C01810=1159.074,186.001,-60.182,-178.162,7.026,148.772
C01811=1159.078,185.752,-60.160,-178.165,7.023,148.772
C01812=1159.083,185.503,-60.136,-178.168,7.021,148.772
C01813=1159.087,185.254,-60.113,-178.170,7.019,148.772
C01814=1159.092,185.005,-60.089,-178.174,7.017,148.773
C01815=1159.097,184.757,-60.067,-178.176,7.015,148.773
C01816=1159.101,184.508,-60.044,-178.178,7.013,148.773
C01817=1159.107,184.238,-60.019,-178.182,7.010,148.774
C01818=1159.112,183.969,-59.994,-178.185,7.008,148.774
C01819=1159.117,183.699,-59.969,-178.187,7.006,148.774
C01820=1159.121,183.429,-59.943,-178.190,7.003,148.774
C01821=1159.127,183.180,-59.921,-178.193,7.001,148.775
C01822=1159.131,182.932,-59.898,-178.196,6.999,148.775
C01823=1159.135,182.683,-59.875,-178.199,6.997,148.775
C01824=1159.140,182.433,-59.851,-178.201,6.995,148.776
C01825=1159.144,182.185,-59.829,-178.205,6.992,148.776
C01826=1159.149,181.936,-59.806,-178.207,6.991,148.776
C01827=1159.154,181.687,-59.783,-178.209,6.989,148.776
C01828=1159.158,181.438,-59.760,-178.212,6.987,148.777
C01829=1159.163,181.189,-59.737,-178.215,6.984,148.777
C01830=1159.168,180.940,-59.713,-178.218,6.982,148.777
C01831=1159.172,180.692,-59.691,-178.220,6.980,148.778
C01832=1159.177,180.442,-59.668,-178.224,6.978,148.778
C01833=1159.181,180.194,-59.646,-178.226,6.976,148.778
C01834=1159.186,179.945,-59.622,-178.229,6.974,148.778
C01835=1159.190,179.697,-59.600,-178.232,6.971,148.779
C01836=1159.195,179.447,-59.577,-178.234,6.970,148.779
C01837=1159.200,179.198,-59.554,-178.237,6.968,148.780
C01838=1159.204,178.949,-59.531,-178.240,6.965,148.780
C01839=1159.210,178.700,-59.509,-178.243,6.963,148.780
C01840=1159.214,178.451,-59.486,-178.245,6.961,148.780
C01841=1159.218,178.202,-59.463,-178.248,6.960,148.781
C01842=1159.223,177.953,-59.441,-178.251,6.957,148.781
C01843=1159.228,177.705,-59.418,-178.254,6.955,148.781
C01844=1159.232,177.455,-59.396,-178.256,6.953,148.782
C01845=1159.237,177.206,-59.372,-178.259,6.951,148.782
C01846=1159.241,176.958,-59.349,-178.262,6.949,148.782
C01847=1159.246,176.709,-59.327,-178.264,6.947,148.782
C01848=1159.250,176.460,-59.304,-178.268,6.944,148.783
C01849=1159.255,176.210,-59.282,-178.270,6.943,148.783
C01850=1159.260,175.962,-59.259,-178.273,6.940,148.783
C01851=1159.265,175.713,-59.237,-178.275,6.939,148.784
C01852=1159.269,175.464,-59.214,-178.278,6.936,148.784
C01853=1159.275,175.215,-59.192,-178.281,6.934,148.784
C01854=1159.278,174.966,-59.169,-178.284,6.933,148.785
C01855=1159.283,174.717,-59.147,-178.286,6.931,148.785
C01856=1159.288,174.469,-59.124,-178.289,6.928,148.785
C01857=1159.292,174.219,-59.102,-178.292,6.926,148.786
C01858=1159.297,173.970,-59.079,-178.295,6.924,148.786
C01859=1159.302,173.722,-59.057,-178.298,6.922,148.786
C01860=1159.306,173.472,-59.035,-178.300,6.920,148.786
C01861=1159.311,173.224,-59.012,-178.303,6.918,148.787
C01862=1159.316,172.975,-58.990,-178.306,6.916,148.787
C01863=1159.320,172.726,-58.966,-178.309,6.914,148.788
C01864=1159.325,172.477,-58.945,-178.311,6.912,148.788
C01865=1159.330,172.228,-58.923,-178.314,6.910,148.788
C01866=1159.334,171.979,-58.899,-178.316,6.908,148.788
C01867=1159.339,171.730,-58.878,-178.320,6.906,148.789
C01868=1159.343,171.481,-58.856,-178.322,6.904,148.789
C01869=1159.349,171.232,-58.833,-178.325,6.902,148.789
C01870=1159.353,170.983,-58.811,-178.327,6.900,148.790
C01871=1159.358,170.734,-58.789,-178.331,6.897,148.790
C01872=1159.363,170.485,-58.766,-178.333,6.896,148.790
C01873=1159.367,170.236,-58.743,-178.336,6.894,148.791
C01874=1159.372,169.987,-58.722,-178.338,6.892,148.791
C01875=1159.376,169.738,-58.700,-178.341,6.890,148.791
C01876=1159.382,169.489,-58.677,-178.344,6.888,148.792
C01877=1159.386,169.240,-58.655,-178.347,6.886,148.792
C01878=1159.390,168.992,-58.633,-178.350,6.884,148.792
C01879=1159.395,168.742,-58.611,-178.352,6.882,148.793
C01880=1159.400,168.493,-58.589,-178.355,6.879,148.793
C01881=1159.405,168.244,-58.567,-178.358,6.878,148.793
C01882=1159.409,167.996,-58.544,-178.360,6.876,148.794
C01883=1159.413,167.747,-58.522,-178.363,6.874,148.794
C01884=1159.419,167.498,-58.500,-178.366,6.872,148.794
C01885=1159.423,167.248,-58.478,-178.369,6.870,148.795
C01886=1159.428,167.000,-58.456,-178.371,6.868,148.795
C01887=1159.432,166.750,-58.434,-178.374,6.866,148.795
C01888=1159.437,166.502,-58.412,-178.377,6.864,148.796
C01889=1159.442,166.252,-58.390,-178.380,6.862,148.796
C01890=1159.447,166.003,-58.368,-178.383,6.860,148.796
C01891=1159.451,165.754,-58.346,-178.385,6.858,148.797
C01892=1159.456,165.505,-58.324,-178.388,6.856,148.797
C01893=1159.461,165.256,-58.302,-178.390,6.854,148.797
C01894=1159.465,165.007,-58.281,-178.394,6.852,148.798
C01895=1159.470,164.758,-58.259,-178.396,6.850,148.798
C01896=1159.475,164.509,-58.237,-178.399,6.848,148.798
C01897=1159.479,164.260,-58.215,-178.402,6.847,148.799
C01898=1159.484,164.011,-58.193,-178.404,6.845,148.799
C01899=1159.489,163.762,-58.171,-178.407,6.842,148.799
C01900=1159.494,163.513,-58.149,-178.410,6.840,148.800
C01901=1159.498,163.264,-58.127,-178.413,6.838,148.800
C01902=1159.503,163.015,-58.105,-178.415,6.837,148.800
C01903=1159.508,162.767,-58.083,-178.418,6.835,148.801
C01904=1159.512,162.517,-58.061,-178.421,6.833,148.801
C01905=1159.517,162.269,-58.040,-178.424,6.831,148.801
C01906=1159.521,162.019,-58.018,-178.427,6.829,148.802
C01907=1159.526,161.771,-57.996,-178.429,6.827,148.802
C01908=1159.531,161.522,-57.974,-178.432,6.825,148.802
C01909=1159.535,161.272,-57.953,-178.434,6.823,148.803
C01910=1159.540,161.023,-57.931,-178.437,6.821,148.803
C01911=1159.544,160.774,-57.909,-178.440,6.819,148.803
C01912=1159.549,160.525,-57.888,-178.443,6.817,148.804
C01913=1159.554,160.277,-57.866,-178.446,6.816,148.804
C01914=1159.559,160.027,-57.845,-178.448,6.814,148.805
C01915=1159.564,159.778,-57.823,-178.451,6.812,148.805
C01916=1159.568,159.529,-57.801,-178.453,6.810,148.805
C01917=1159.573,159.280,-57.779,-178.456,6.807,148.805
C01918=1159.578,159.031,-57.758,-178.459,6.806,148.806
C01919=1159.582,158.783,-57.737,-178.462,6.804,148.806
C01920=1159.586,158.533,-57.715,-178.465,6.802,148.807
C01921=1159.592,158.264,-57.692,-178.467,6.800,148.807
C01922=1159.596,157.995,-57.668,-178.471,6.798,148.807
C01923=1159.602,157.726,-57.645,-178.473,6.796,148.808
C01924=1159.607,157.458,-57.622,-178.477,6.794,148.808
C01925=1159.611,157.208,-57.600,-178.479,6.792,148.808
C01926=1159.616,156.959,-57.579,-178.482,6.790,148.809
C01927=1159.621,156.710,-57.558,-178.485,6.788,148.809
C01928=1159.626,156.461,-57.536,-178.487,6.787,148.809
C01929=1159.631,156.212,-57.515,-178.490,6.785,148.810
C01930=1159.636,155.963,-57.493,-178.493,6.782,148.810
C01931=1159.640,155.714,-57.472,-178.496,6.781,148.811
C01932=1159.644,155.465,-57.451,-178.499,6.779,148.811
C01933=1159.649,155.216,-57.429,-178.501,6.777,148.811
C01934=1159.654,154.967,-57.408,-178.504,6.775,148.812
C01935=1159.659,154.718,-57.386,-178.506,6.773,148.812
C01936=1159.663,154.469,-57.366,-178.509,6.772,148.812
C01937=1159.668,154.220,-57.344,-178.512,6.770,148.813
C01938=1159.673,153.971,-57.323,-178.514,6.768,148.813
C01939=1159.677,153.722,-57.301,-178.518,6.766,148.813
C01940=1159.683,153.472,-57.280,-178.520,6.764,148.814
C01941=1159.687,153.224,-57.259,-178.523,6.762,148.814
C01942=1159.692,152.975,-57.238,-178.526,6.760,148.815
C01943=1159.697,152.726,-57.216,-178.528,6.759,148.815
C01944=1159.701,152.476,-57.195,-178.531,6.757,148.815
C01945=1159.706,152.227,-57.174,-178.534,6.755,148.816
C01946=1159.711,151.978,-57.153,-178.537,6.753,148.816
C01947=1159.716,151.729,-57.132,-178.539,6.752,148.816
C01948=1159.720,151.481,-57.111,-178.543,6.749,148.817
C01949=1159.725,151.231,-57.089,-178.545,6.747,148.817
C01950=1159.730,150.982,-57.068,-178.548,6.746,148.818
C01951=1159.735,150.733,-57.047,-178.551,6.744,148.818
C01952=1159.739,150.484,-57.026,-178.553,6.742,148.818
C01953=1159.744,150.235,-57.005,-178.556,6.740,148.819
C01954=1159.748,149.985,-56.983,-178.559,6.739,148.819
C01955=1159.753,149.737,-56.963,-178.561,6.737,148.819
C01956=1159.758,149.487,-56.942,-178.564,6.735,148.820
C01957=1159.762,149.239,-56.921,-178.566,6.733,148.820
C01958=1159.767,148.990,-56.900,-178.569,6.731,148.820
C01959=1159.773,148.740,-56.879,-178.572,6.729,148.821
C01960=1159.777,148.492,-56.858,-178.575,6.727,148.821
C01961=1159.781,148.242,-56.837,-178.578,6.725,148.822
C01962=1159.786,147.993,-56.816,-178.581,6.724,148.822
C01963=1159.791,147.744,-56.795,-178.583,6.722,148.822
C01964=1159.796,147.495,-56.774,-178.586,6.720,148.823
C01965=1159.800,147.246,-56.753,-178.589,6.719,148.823
C01966=1159.805,146.997,-56.732,-178.591,6.717,148.823
C01967=1159.810,146.748,-56.712,-178.594,6.715,148.824
C01968=1159.815,146.499,-56.691,-178.597,6.713,148.824
C01969=1159.819,146.250,-56.670,-178.599,6.712,148.825
C01970=1159.824,146.001,-56.648,-178.602,6.710,148.825
C01971=1159.829,145.751,-56.627,-178.605,6.708,148.825
C01972=1159.833,145.502,-56.607,-178.608,6.706,148.826
C01973=1159.838,145.253,-56.586,-178.610,6.705,148.826
C01974=1159.843,145.004,-56.566,-178.613,6.703,148.827
C01975=1159.848,144.755,-56.545,-178.616,6.700,148.827
C01976=1159.853,144.506,-56.524,-178.619,6.699,148.827
C01977=1159.858,144.257,-56.503,-178.622,6.697,148.828
C01978=1159.862,144.008,-56.483,-178.624,6.695,148.828
C01979=1159.867,143.759,-56.463,-178.627,6.693,148.828
C01980=1159.872,143.510,-56.442,-178.630,6.692,148.829
C01981=1159.876,143.261,-56.421,-178.632,6.690,148.829
C01982=1159.881,143.011,-56.400,-178.635,6.688,148.830
C01983=1159.886,142.762,-56.380,-178.638,6.687,148.830
C01984=1159.891,142.513,-56.359,-178.641,6.685,148.830
C01985=1159.895,142.264,-56.339,-178.643,6.683,148.831
C01986=1159.900,142.015,-56.318,-178.646,6.681,148.831
C01987=1159.905,141.766,-56.297,-178.649,6.680,148.832
C01988=1159.909,141.517,-56.277,-178.651,6.678,148.832
C01989=1159.915,141.268,-56.256,-178.654,6.676,148.832
C01990=1159.919,141.019,-56.236,-178.657,6.674,148.833
C01991=1159.923,140.770,-56.215,-178.660,6.673,148.833
C01992=1159.929,140.521,-56.194,-178.662,6.671,148.833
C01993=1159.933,140.272,-56.174,-178.665,6.670,148.834
C01994=1159.938,140.023,-56.154,-178.668,6.668,148.834
C01995=1159.943,139.773,-56.133,-178.671,6.666,148.835
C01996=1159.947,139.524,-56.113,-178.674,6.664,148.835
C01997=1159.952,139.275,-56.093,-178.676,6.663,148.836
C01998=1159.957,139.026,-56.072,-178.679,6.661,148.836
C01999=1159.962,138.777,-56.051,-178.682,6.659,148.836
C02000=1159.966,138.528,-56.031,-178.684,6.658,148.837
C02001=1159.971,138.278,-56.010,-178.687,6.656,148.837
C02002=1159.976,138.029,-55.990,-178.690,6.654,148.838
C02003=1159.980,137.780,-55.970,-178.692,6.652,148.838
C02004=1159.985,137.531,-55.949,-178.695,6.651,148.838
C02005=1159.990,137.282,-55.928,-178.698,6.649,148.839
C02006=1159.995,137.032,-55.909,-178.701,6.647,148.839
C02007=1159.999,136.783,-55.888,-178.703,6.645,148.840
C02008=1160.004,136.534,-55.868,-178.706,6.644,148.840
C02009=1160.009,136.286,-55.847,-178.709,6.642,148.840
C02010=1160.014,136.036,-55.828,-178.711,6.640,148.841
C02011=1160.018,135.787,-55.807,-178.714,6.639,148.841
C02012=1160.023,135.538,-55.787,-178.717,6.637,148.841
C02013=1160.028,135.288,-55.767,-178.720,6.635,148.842
C02014=1160.033,135.039,-55.746,-178.723,6.634,148.842
C02015=1160.037,134.791,-55.726,-178.725,6.632,148.843
C02016=1160.042,134.541,-55.706,-178.728,6.630,148.843
C02017=1160.047,134.293,-55.686,-178.731,6.629,148.844
C02018=1160.052,134.043,-55.665,-178.734,6.627,148.844
C02019=1160.057,133.794,-55.646,-178.736,6.625,148.844
C02020=1160.061,133.545,-55.625,-178.739,6.623,148.845
C02021=1160.066,133.295,-55.606,-178.742,6.622,148.845
C02022=1160.071,133.046,-55.585,-178.744,6.620,148.846
C02023=1160.075,132.797,-55.566,-178.747,6.618,148.846
C02024=1160.081,132.548,-55.545,-178.750,6.616,148.846
C02025=1160.086,132.280,-55.524,-178.753,6.615,148.847
C02026=1160.091,132.012,-55.502,-178.756,6.613,148.847
C02027=1160.096,131.743,-55.481,-178.758,6.612,148.848
C02028=1160.101,131.474,-55.460,-178.761,6.610,148.848
C02029=1160.106,131.225,-55.439,-178.764,6.608,148.849
C02030=1160.110,130.975,-55.419,-178.767,6.607,148.849
C02031=1160.116,130.726,-55.399,-178.770,6.605,148.850
C02032=1160.121,130.477,-55.379,-178.772,6.603,148.850
C02033=1160.125,130.228,-55.359,-178.775,6.602,148.850
C02034=1160.130,129.979,-55.339,-178.778,6.600,148.851
C02035=1160.135,129.730,-55.319,-178.781,6.598,148.851
C02036=1160.139,129.480,-55.299,-178.783,6.597,148.852
C02037=1160.145,129.231,-55.280,-178.786,6.595,148.852
C02038=1160.149,128.982,-55.259,-178.789,6.593,148.852
C02039=1160.154,128.733,-55.240,-178.791,6.591,148.853
C02040=1160.159,128.483,-55.220,-178.795,6.590,148.853
C02041=1160.164,128.235,-55.200,-178.797,6.588,148.854
C02042=1160.168,127.986,-55.181,-178.800,6.587,148.854
C02043=1160.173,127.737,-55.160,-178.803,6.585,148.855
C02044=1160.177,127.487,-55.140,-178.805,6.584,148.855
C02045=1160.183,127.238,-55.121,-178.808,6.582,148.855
C02046=1160.188,126.989,-55.102,-178.810,6.581,148.856
C02047=1160.192,126.740,-55.081,-178.813,6.579,148.856
C02048=1160.197,126.491,-55.062,-178.816,6.577,148.857
C02049=1160.202,126.241,-55.042,-178.819,6.576,148.857
C02050=1160.207,125.992,-55.022,-178.822,6.574,148.858
C02051=1160.211,125.743,-55.003,-178.824,6.572,148.858
C02052=1160.216,125.494,-54.984,-178.827,6.571,148.858
C02053=1160.221,125.245,-54.964,-178.830,6.569,148.859
C02054=1160.225,124.996,-54.943,-178.832,6.567,148.859
C02055=1160.230,124.747,-54.924,-178.835,6.566,148.860
C02056=1160.235,124.497,-54.905,-178.838,6.565,148.860
C02057=1160.240,124.248,-54.885,-178.840,6.563,148.861
C02058=1160.245,123.999,-54.866,-178.843,6.561,148.861
C02059=1160.250,123.749,-54.846,-178.846,6.560,148.861
C02060=1160.254,123.501,-54.826,-178.849,6.558,148.862
C02061=1160.259,123.252,-54.807,-178.851,6.556,148.862
C02062=1160.264,123.002,-54.787,-178.854,6.555,148.863
C02063=1160.269,122.753,-54.768,-178.857,6.553,148.863
C02064=1160.274,122.504,-54.748,-178.860,6.551,148.864
C02065=1160.279,122.254,-54.729,-178.862,6.551,148.864
C02066=1160.283,122.005,-54.710,-178.865,6.549,148.864
C02067=1160.288,121.756,-54.690,-178.868,6.547,148.865
C02068=1160.293,121.506,-54.671,-178.870,6.545,148.865
C02069=1160.298,121.258,-54.651,-178.873,6.544,148.866
C02070=1160.302,121.009,-54.631,-178.876,6.542,148.866
C02071=1160.306,120.759,-54.612,-178.879,6.541,148.867
C02072=1160.312,120.510,-54.593,-178.882,6.539,148.867
C02073=1160.317,120.261,-54.573,-178.884,6.538,148.867
C02074=1160.322,120.012,-54.554,-178.886,6.536,148.868
C02075=1160.326,119.763,-54.535,-178.889,6.535,148.868
C02076=1160.331,119.513,-54.515,-178.892,6.533,148.869
C02077=1160.336,119.264,-54.496,-178.895,6.532,148.869
C02078=1160.341,119.015,-54.476,-178.898,6.530,148.870
C02079=1160.345,118.766,-54.457,-178.900,6.528,148.870
C02080=1160.350,118.516,-54.438,-178.903,6.527,148.870
C02081=1160.356,118.267,-54.419,-178.905,6.525,148.871
C02082=1160.360,118.018,-54.400,-178.909,6.524,148.871
C02083=1160.365,117.769,-54.381,-178.911,6.522,148.872
C02084=1160.370,117.519,-54.361,-178.914,6.521,148.872
C02085=1160.374,117.270,-54.342,-178.917,6.519,148.873
C02086=1160.379,117.021,-54.323,-178.919,6.517,148.873
C02087=1160.384,116.772,-54.303,-178.922,6.516,148.874
C02088=1160.389,116.523,-54.284,-178.925,6.515,148.874
C02089=1160.394,116.273,-54.265,-178.927,6.513,148.875
C02090=1160.399,116.024,-54.246,-178.930,6.512,148.875
C02091=1160.403,115.775,-54.227,-178.933,6.510,148.875
C02092=1160.408,115.526,-54.208,-178.936,6.508,148.876
C02093=1160.413,115.276,-54.188,-178.938,6.508,148.876
C02094=1160.418,115.028,-54.169,-178.941,6.506,148.877
C02095=1160.423,114.778,-54.150,-178.944,6.504,148.877
C02096=1160.427,114.529,-54.132,-178.946,6.502,148.878
C02097=1160.432,114.280,-54.112,-178.949,6.501,148.878
C02098=1160.437,114.031,-54.093,-178.952,6.499,148.879
C02099=1160.442,113.781,-54.074,-178.954,6.499,148.879
C02100=1160.447,113.532,-54.055,-178.957,6.497,148.879
C02101=1160.452,113.283,-54.036,-178.960,6.495,148.880
C02102=1160.457,113.033,-54.018,-178.963,6.493,148.880
C02103=1160.461,112.785,-53.999,-178.966,6.492,148.881
C02104=1160.466,112.535,-53.979,-178.968,6.490,148.881
C02105=1160.472,112.286,-53.961,-178.971,6.489,148.882
C02106=1160.476,112.036,-53.942,-178.973,6.488,148.882
C02107=1160.481,111.787,-53.922,-178.976,6.486,148.883
C02108=1160.485,111.538,-53.904,-178.979,6.485,148.883
C02109=1160.491,111.289,-53.885,-178.982,6.483,148.884
C02110=1160.495,111.040,-53.866,-178.984,6.482,148.884
C02111=1160.500,110.790,-53.847,-178.987,6.480,148.884
C02112=1160.505,110.541,-53.828,-178.990,6.479,148.885
C02113=1160.510,110.291,-53.809,-178.993,6.477,148.885
C02114=1160.515,110.043,-53.791,-178.995,6.476,148.886
C02115=1160.519,109.794,-53.772,-178.998,6.475,148.886
C02116=1160.524,109.544,-53.753,-179.000,6.473,148.887
C02117=1160.529,109.295,-53.734,-179.004,6.472,148.887
C02118=1160.534,109.045,-53.715,-179.006,6.470,148.888
C02119=1160.539,108.797,-53.697,-179.009,6.468,148.888
C02120=1160.544,108.547,-53.678,-179.011,6.467,148.888
C02121=1160.548,108.298,-53.659,-179.014,6.466,148.889
C02122=1160.553,108.049,-53.641,-179.017,6.464,148.890
C02123=1160.558,107.800,-53.622,-179.020,6.463,148.890
C02124=1160.563,107.550,-53.603,-179.022,6.462,148.890
C02125=1160.568,107.301,-53.584,-179.025,6.460,148.891
C02126=1160.572,107.051,-53.566,-179.028,6.459,148.891
C02127=1160.577,106.803,-53.547,-179.031,6.457,148.892
C02128=1160.583,106.553,-53.529,-179.033,6.455,148.892
C02129=1160.588,106.285,-53.509,-179.036,6.454,148.893
C02130=1160.593,106.016,-53.488,-179.039,6.452,148.893
C02131=1160.598,105.748,-53.469,-179.042,6.450,148.894
C02132=1160.604,105.479,-53.449,-179.045,6.449,148.894
C02133=1160.608,105.230,-53.430,-179.047,6.448,148.895
C02134=1160.612,104.981,-53.412,-179.050,6.447,148.895
C02135=1160.618,104.732,-53.393,-179.053,6.445,148.896
C02136=1160.623,104.483,-53.374,-179.056,6.443,148.896
C02137=1160.627,104.233,-53.356,-179.058,6.443,148.897
C02138=1160.633,103.984,-53.337,-179.061,6.441,148.897
C02139=1160.637,103.735,-53.319,-179.063,6.439,148.897
C02140=1160.642,103.485,-53.300,-179.067,6.438,148.898
C02141=1160.647,103.236,-53.282,-179.069,6.437,148.898
C02142=1160.652,102.987,-53.263,-179.071,6.435,148.899
C02143=1160.657,102.738,-53.245,-179.075,6.434,148.900
C02144=1160.661,102.488,-53.227,-179.077,6.432,148.900
C02145=1160.667,102.239,-53.208,-179.080,6.431,148.900
C02146=1160.671,101.990,-53.189,-179.082,6.430,148.901
C02147=1160.676,101.741,-53.172,-179.085,6.428,148.901
C02148=1160.681,101.491,-53.153,-179.088,6.427,148.902
C02149=1160.685,101.242,-53.135,-179.090,6.426,148.902
C02150=1160.691,100.993,-53.116,-179.093,6.424,148.903
C02151=1160.696,100.744,-53.098,-179.096,6.423,148.903
C02152=1160.700,100.494,-53.080,-179.098,6.422,148.904
C02153=1160.705,100.245,-53.062,-179.101,6.420,148.904
C02154=1160.710,99.996,-53.044,-179.104,6.418,148.905
C02155=1160.716,99.746,-53.025,-179.107,6.417,148.905
C02156=1160.720,99.498,-53.006,-179.109,6.416,148.906
C02157=1160.724,99.248,-52.988,-179.112,6.414,148.906
C02158=1160.729,98.998,-52.970,-179.115,6.413,148.907
C02159=1160.734,98.749,-52.952,-179.118,6.411,148.907
C02160=1160.739,98.500,-52.934,-179.120,6.410,148.907
C02161=1160.744,98.251,-52.916,-179.123,6.409,148.908
C02162=1160.749,98.001,-52.897,-179.126,6.407,148.909
C02163=1160.754,97.752,-52.879,-179.128,6.407,148.909
C02164=1160.759,97.502,-52.861,-179.131,6.405,148.909
C02165=1160.764,97.253,-52.843,-179.134,6.404,148.910
C02166=1160.769,97.004,-52.825,-179.136,6.403,148.910
C02167=1160.774,96.755,-52.807,-179.139,6.401,148.911
C02168=1160.778,96.505,-52.789,-179.142,6.399,148.911
C02169=1160.783,96.256,-52.771,-179.145,6.398,148.912
C02170=1160.788,96.007,-52.753,-179.147,6.397,148.912
C02171=1160.793,95.757,-52.735,-179.150,6.395,148.913
C02172=1160.798,95.508,-52.717,-179.153,6.394,148.913
C02173=1160.803,95.259,-52.699,-179.155,6.393,148.914
C02174=1160.807,95.010,-52.681,-179.158,6.391,148.914
C02175=1160.812,94.761,-52.663,-179.160,6.390,148.915
C02176=1160.817,94.511,-52.645,-179.163,6.389,148.915
C02177=1160.822,94.261,-52.626,-179.166,6.387,148.916
C02178=1160.827,94.012,-52.608,-179.169,6.386,148.916
C02179=1160.832,93.763,-52.590,-179.172,6.384,148.917
C02180=1160.837,93.514,-52.572,-179.174,6.384,148.917
C02181=1160.842,93.265,-52.554,-179.177,6.382,148.918
C02182=1160.846,93.016,-52.537,-179.180,6.381,148.918
C02183=1160.851,92.766,-52.520,-179.182,6.380,148.919
C02184=1160.856,92.517,-52.502,-179.185,6.378,148.919
C02185=1160.861,92.268,-52.484,-179.187,6.376,148.919
C02186=1160.866,92.019,-52.466,-179.190,6.376,148.920
C02187=1160.870,91.769,-52.447,-179.193,6.374,148.921
C02188=1160.875,91.519,-52.429,-179.195,6.372,148.921
C02189=1160.881,91.270,-52.412,-179.198,6.372,148.922
C02190=1160.885,91.021,-52.394,-179.201,6.370,148.922
C02191=1160.890,90.771,-52.376,-179.204,6.368,148.922
C02192=1160.895,90.522,-52.358,-179.206,6.368,148.923
C02193=1160.901,90.272,-52.341,-179.209,6.366,148.924
C02194=1160.905,90.023,-52.323,-179.212,6.364,148.924
C02195=1160.910,89.774,-52.305,-179.214,6.364,148.925
C02196=1160.915,89.525,-52.287,-179.217,6.362,148.925
C02197=1160.920,89.275,-52.270,-179.220,6.361,148.925
C02198=1160.925,89.026,-52.252,-179.222,6.360,148.926
C02199=1160.930,88.777,-52.234,-179.225,6.358,148.926
C02200=1160.935,88.527,-52.217,-179.227,6.357,148.927
C02201=1160.940,88.278,-52.199,-179.230,6.356,148.928
C02202=1160.945,88.029,-52.181,-179.233,6.354,148.928
C02203=1160.949,87.779,-52.164,-179.235,6.354,148.928
C02204=1160.954,87.530,-52.146,-179.239,6.352,148.929
C02205=1160.959,87.281,-52.128,-179.241,6.351,148.929
C02206=1160.964,87.031,-52.111,-179.243,6.350,148.930
C02207=1160.969,86.782,-52.093,-179.247,6.348,148.931
C02208=1160.973,86.533,-52.076,-179.249,6.347,148.931
C02209=1160.978,86.283,-52.058,-179.251,6.346,148.931
C02210=1160.983,86.034,-52.041,-179.255,6.344,148.932
C02211=1160.989,85.784,-52.023,-179.257,6.344,148.932
C02212=1160.993,85.535,-52.005,-179.260,6.342,148.933
C02213=1160.998,85.286,-51.988,-179.263,6.341,148.934
C02214=1161.003,85.037,-51.971,-179.265,6.340,148.934
C02215=1161.008,84.787,-51.953,-179.268,6.338,148.934
C02216=1161.014,84.538,-51.936,-179.271,6.337,148.935
C02217=1161.018,84.289,-51.918,-179.273,6.336,148.935
C02218=1161.023,84.040,-51.901,-179.276,6.334,148.936
C02219=1161.028,83.790,-51.883,-179.278,6.334,148.937
C02220=1161.033,83.541,-51.866,-179.281,6.332,148.937
C02221=1161.037,83.292,-51.848,-179.284,6.330,148.937
C02222=1161.042,83.042,-51.831,-179.286,6.330,148.938
C02223=1161.047,82.793,-51.813,-179.289,6.328,148.938
C02224=1161.052,82.543,-51.797,-179.292,6.327,148.939
C02225=1161.057,82.294,-51.779,-179.295,6.326,148.940
C02226=1161.062,82.044,-51.761,-179.297,6.324,148.940
C02227=1161.067,81.796,-51.745,-179.300,6.324,148.941
C02228=1161.072,81.546,-51.727,-179.303,6.322,148.941
C02229=1161.077,81.297,-51.710,-179.305,6.321,148.941
C02230=1161.081,81.048,-51.692,-179.308,6.320,148.942
C02231=1161.087,80.798,-51.675,-179.311,6.318,148.943
C02232=1161.092,80.548,-51.658,-179.313,6.317,148.943
C02233=1161.097,80.280,-51.640,-179.316,6.316,148.944
C02234=1161.102,80.012,-51.621,-179.319,6.314,148.944
C02235=1161.108,79.743,-51.602,-179.322,6.313,148.945
C02236=1161.113,79.475,-51.584,-179.325,6.312,148.945
C02237=1161.118,79.226,-51.567,-179.327,6.311,148.946
C02238=1161.123,78.976,-51.549,-179.330,6.309,148.946
C02239=1161.127,78.727,-51.532,-179.333,6.308,148.947
C02240=1161.133,78.477,-51.515,-179.335,6.307,148.947
C02241=1161.137,78.228,-51.498,-179.338,6.306,148.948
C02242=1161.143,77.979,-51.481,-179.341,6.305,148.948
C02243=1161.147,77.730,-51.464,-179.343,6.304,148.949
C02244=1161.152,77.480,-51.447,-179.346,6.302,148.949
C02245=1161.157,77.231,-51.429,-179.349,6.301,148.950
C02246=1161.162,76.981,-51.412,-179.351,6.300,148.950
C02247=1161.168,76.732,-51.395,-179.354,6.298,148.951
C02248=1161.172,76.483,-51.379,-179.356,6.298,148.951
C02249=1161.177,76.233,-51.361,-179.359,6.296,148.952
C02250=1161.181,75.984,-51.344,-179.362,6.295,148.952
C02251=1161.187,75.734,-51.327,-179.365,6.294,148.953
C02252=1161.192,75.485,-51.310,-179.367,6.293,148.954
C02253=1161.197,75.236,-51.293,-179.370,6.291,148.954
C02254=1161.201,74.986,-51.277,-179.373,6.290,148.954
C02255=1161.206,74.737,-51.260,-179.375,6.289,148.955
C02256=1161.211,74.488,-51.242,-179.378,6.288,148.955
C02257=1161.216,74.239,-51.226,-179.381,6.287,148.956
C02258=1161.221,73.989,-51.208,-179.383,6.285,148.957
C02259=1161.226,73.739,-51.192,-179.386,6.285,148.957
C02260=1161.231,73.490,-51.175,-179.389,6.283,148.958
C02261=1161.236,73.241,-51.158,-179.391,6.282,148.958
C02262=1161.241,72.991,-51.141,-179.394,6.281,148.959
C02263=1161.246,72.742,-51.124,-179.397,6.279,148.959
C02264=1161.251,72.493,-51.108,-179.399,6.278,148.960
C02265=1161.256,72.243,-51.091,-179.402,6.277,148.960
C02266=1161.260,71.993,-51.074,-179.404,6.276,148.961
C02267=1161.266,71.744,-51.057,-179.408,6.275,148.961
C02268=1161.271,71.495,-51.040,-179.410,6.274,148.962
C02269=1161.275,71.245,-51.024,-179.412,6.272,148.962
C02270=1161.281,70.996,-51.007,-179.415,6.272,148.963
C02271=1161.285,70.747,-50.990,-179.418,6.270,148.963
C02272=1161.290,70.497,-50.973,-179.420,6.270,148.964
C02273=1161.296,70.248,-50.957,-179.423,6.268,148.964
C02274=1161.300,69.999,-50.940,-179.425,6.267,148.965
C02275=1161.305,69.749,-50.923,-179.429,6.266,148.965
C02276=1161.311,69.500,-50.906,-179.431,6.265,148.966
C02277=1161.315,69.251,-50.890,-179.434,6.264,148.967
C02278=1161.320,69.001,-50.872,-179.436,6.263,148.967
C02279=1161.325,68.752,-50.856,-179.439,6.261,148.967
C02280=1161.330,68.503,-50.839,-179.441,6.261,148.968
C02281=1161.334,68.253,-50.823,-179.444,6.259,148.969
C02282=1161.340,68.004,-50.806,-179.447,6.258,148.969
C02283=1161.345,67.754,-50.790,-179.450,6.257,148.970
C02284=1161.349,67.504,-50.773,-179.452,6.256,148.970
C02285=1161.355,67.255,-50.756,-179.455,6.255,148.971
C02286=1161.360,67.006,-50.740,-179.457,6.254,148.971
C02287=1161.364,66.756,-50.723,-179.460,6.252,148.972
C02288=1161.369,66.508,-50.707,-179.462,6.252,148.972
C02289=1161.374,66.258,-50.691,-179.466,6.250,148.973
C02290=1161.380,66.008,-50.674,-179.468,6.249,148.973
C02291=1161.384,65.759,-50.657,-179.471,6.248,148.974
C02292=1161.389,65.509,-50.640,-179.473,6.247,148.974
C02293=1161.394,65.261,-50.624,-179.476,6.246,148.975
C02294=1161.399,65.010,-50.608,-179.479,6.245,148.976
C02295=1161.404,64.761,-50.591,-179.481,6.243,148.976
C02296=1161.409,64.512,-50.575,-179.484,6.243,148.977
C02297=1161.414,64.263,-50.559,-179.487,6.241,148.977
C02298=1161.419,64.013,-50.542,-179.489,6.240,148.977
C02299=1161.424,63.763,-50.525,-179.492,6.239,148.978
C02300=1161.429,63.515,-50.509,-179.494,6.238,148.979
C02301=1161.434,63.264,-50.493,-179.497,6.237,148.979
C02302=1161.439,63.016,-50.477,-179.500,6.236,148.980
C02303=1161.443,62.766,-50.460,-179.503,6.235,148.980
C02304=1161.449,62.517,-50.444,-179.505,6.234,148.981
C02305=1161.453,62.267,-50.428,-179.508,6.232,148.981
C02306=1161.459,62.018,-50.411,-179.510,6.232,148.982
C02307=1161.464,61.768,-50.395,-179.513,6.230,148.982
C02308=1161.469,61.519,-50.378,-179.516,6.229,148.983
C02309=1161.473,61.270,-50.362,-179.518,6.229,148.983
C02310=1161.478,61.020,-50.346,-179.521,6.227,148.984
C02311=1161.483,60.771,-50.330,-179.523,6.226,148.985
C02312=1161.488,60.521,-50.314,-179.526,6.225,148.985
C02313=1161.493,60.272,-50.297,-179.529,6.224,148.986
C02314=1161.498,60.022,-50.281,-179.531,6.223,148.986
C02315=1161.503,59.773,-50.265,-179.534,6.222,148.987
C02316=1161.508,59.524,-50.248,-179.537,6.220,148.987
C02317=1161.514,59.274,-50.232,-179.539,6.220,148.988
C02318=1161.519,59.025,-50.216,-179.542,6.218,148.988
C02319=1161.524,58.775,-50.200,-179.545,6.218,148.989
C02320=1161.529,58.526,-50.184,-179.547,6.217,148.989
C02321=1161.533,58.276,-50.168,-179.550,6.215,148.990
C02322=1161.538,58.027,-50.151,-179.552,6.215,148.990
C02323=1161.543,57.777,-50.135,-179.555,6.213,148.991
C02324=1161.548,57.529,-50.119,-179.558,6.213,148.992
C02325=1161.553,57.278,-50.103,-179.560,6.211,148.992
C02326=1161.558,57.030,-50.087,-179.563,6.210,148.993
C02327=1161.563,56.780,-50.071,-179.565,6.209,148.993
C02328=1161.568,56.530,-50.055,-179.568,6.208,148.994
C02329=1161.573,56.281,-50.039,-179.571,6.207,148.994
C02330=1161.578,56.031,-50.023,-179.574,6.206,148.995
C02331=1161.583,55.782,-50.007,-179.576,6.205,148.995
C02332=1161.588,55.532,-49.991,-179.579,6.203,148.996
C02333=1161.594,55.283,-49.975,-179.581,6.203,148.996
C02334=1161.598,55.033,-49.959,-179.583,6.202,148.997
C02335=1161.603,54.784,-49.943,-179.587,6.201,148.998
C02336=1161.608,54.536,-49.927,-179.589,6.200,148.998
C02337=1161.613,54.266,-49.910,-179.592,6.199,148.999
C02338=1161.618,53.998,-49.893,-179.595,6.197,148.999
C02339=1161.624,53.729,-49.876,-179.597,6.196,149.000
C02340=1161.629,53.461,-49.859,-179.601,6.195,149.000
C02341=1161.634,53.211,-49.843,-179.603,6.194,149.001
C02342=1161.640,52.961,-49.827,-179.606,6.193,149.001
C02343=1161.645,52.713,-49.811,-179.608,6.192,149.002
C02344=1161.649,52.463,-49.795,-179.611,6.192,149.003
C02345=1161.655,52.213,-49.779,-179.614,6.190,149.003
C02346=1161.660,51.964,-49.763,-179.616,6.190,149.004
C02347=1161.665,51.714,-49.747,-179.619,6.188,149.004
C02348=1161.669,51.465,-49.732,-179.622,6.187,149.005
C02349=1161.675,51.216,-49.717,-179.624,6.187,149.005
C02350=1161.679,50.966,-49.701,-179.627,6.185,149.006
C02351=1161.685,50.717,-49.684,-179.629,6.184,149.006
C02352=1161.690,50.467,-49.669,-179.632,6.183,149.007
C02353=1161.694,50.218,-49.653,-179.635,6.182,149.007
C02354=1161.699,49.968,-49.638,-179.637,6.181,149.008
C02355=1161.705,49.719,-49.622,-179.640,6.180,149.009
C02356=1161.709,49.469,-49.606,-179.642,6.179,149.009
C02357=1161.715,49.220,-49.590,-179.645,6.179,149.010
C02358=1161.719,48.971,-49.575,-179.648,6.177,149.010
C02359=1161.724,48.721,-49.559,-179.650,6.177,149.011
C02360=1161.729,48.471,-49.543,-179.653,6.175,149.011
C02361=1161.735,48.222,-49.528,-179.656,6.174,149.012
C02362=1161.740,47.972,-49.512,-179.658,6.174,149.012
C02363=1161.744,47.723,-49.496,-179.661,6.172,149.013
C02364=1161.749,47.474,-49.481,-179.663,6.171,149.013
C02365=1161.755,47.225,-49.465,-179.666,6.171,149.014
C02366=1161.759,46.975,-49.450,-179.668,6.169,149.015
C02367=1161.764,46.725,-49.434,-179.671,6.169,149.015
C02368=1161.770,46.476,-49.418,-179.674,6.167,149.016
C02369=1161.774,46.226,-49.402,-179.676,6.167,149.016
C02370=1161.779,45.977,-49.387,-179.679,6.166,149.017
C02371=1161.784,45.727,-49.372,-179.682,6.164,149.017
C02372=1161.790,45.478,-49.356,-179.684,6.164,149.018
C02373=1161.794,45.228,-49.341,-179.687,6.163,149.019
C02374=1161.799,44.979,-49.325,-179.689,6.161,149.019
C02375=1161.805,44.729,-49.310,-179.692,6.161,149.020
C02376=1161.809,44.480,-49.295,-179.694,6.160,149.020
C02377=1161.815,44.231,-49.279,-179.697,6.159,149.021
C02378=1161.819,43.981,-49.263,-179.700,6.158,149.021
C02379=1161.824,43.732,-49.248,-179.702,6.157,149.022
C02380=1161.829,43.482,-49.233,-179.705,6.156,149.022
C02381=1161.835,43.233,-49.217,-179.707,6.155,149.023
C02382=1161.839,42.983,-49.202,-179.710,6.154,149.024
C02383=1161.844,42.734,-49.186,-179.713,6.153,149.024
C02384=1161.850,42.484,-49.171,-179.715,6.152,149.025
C02385=1161.855,42.235,-49.156,-179.717,6.151,149.025
C02386=1161.860,41.985,-49.141,-179.721,6.150,149.026
C02387=1161.865,41.736,-49.126,-179.723,6.149,149.026
C02388=1161.869,41.486,-49.110,-179.725,6.149,149.027
C02389=1161.875,41.237,-49.094,-179.728,6.147,149.027
C02390=1161.879,40.988,-49.079,-179.731,6.147,149.028
C02391=1161.885,40.738,-49.064,-179.733,6.146,149.028
C02392=1161.890,40.489,-49.049,-179.736,6.145,149.029
C02393=1161.895,40.239,-49.034,-179.738,6.144,149.030
C02394=1161.899,39.989,-49.018,-179.741,6.143,149.030
C02395=1161.905,39.740,-49.003,-179.744,6.142,149.031
C02396=1161.910,39.490,-48.987,-179.746,6.141,149.031
C02397=1161.915,39.241,-48.972,-179.749,6.140,149.032
C02398=1161.920,38.991,-48.957,-179.752,6.139,149.032
C02399=1161.925,38.742,-48.942,-179.754,6.138,149.033
C02400=1161.930,38.493,-48.927,-179.757,6.138,149.034
C02401=1161.934,38.243,-48.911,-179.759,6.136,149.034
C02402=1161.940,37.993,-48.896,-179.762,6.135,149.035
C02403=1161.945,37.744,-48.881,-179.764,6.135,149.035
C02404=1161.950,37.495,-48.866,-179.767,6.133,149.036
C02405=1161.955,37.245,-48.851,-179.769,6.133,149.036
C02406=1161.961,36.995,-48.836,-179.772,6.132,149.037
C02407=1161.965,36.746,-48.821,-179.775,6.131,149.038
C02408=1161.971,36.497,-48.805,-179.778,6.130,149.038
C02409=1161.976,36.247,-48.791,-179.780,6.129,149.039
C02410=1161.981,35.998,-48.776,-179.782,6.129,149.039
C02411=1161.986,35.749,-48.761,-179.786,6.127,149.040
C02412=1161.990,35.498,-48.746,-179.788,6.126,149.040
C02413=1161.995,35.249,-48.730,-179.790,6.126,149.041
C02414=1162.000,35.000,-48.715,-179.793,6.124,149.041
C02415=1162.006,34.750,-48.701,-179.796,6.124,149.042
C02416=1162.010,34.501,-48.686,-179.798,6.123,149.043
C02417=1162.016,34.251,-48.671,-179.801,6.122,149.043
C02418=1162.021,34.002,-48.656,-179.803,6.121,149.044
C02419=1162.025,33.752,-48.641,-179.806,6.120,149.044
C02420=1162.031,33.502,-48.626,-179.808,6.120,149.045
C02421=1162.036,33.253,-48.611,-179.811,6.118,149.046
C02422=1162.041,33.004,-48.597,-179.814,6.117,149.046
C02423=1162.046,32.754,-48.581,-179.816,6.117,149.047
C02424=1162.051,32.505,-48.567,-179.818,6.116,149.047
C02425=1162.056,32.255,-48.551,-179.822,6.115,149.048
C02426=1162.061,32.005,-48.537,-179.824,6.114,149.048
C02427=1162.066,31.756,-48.522,-179.826,6.113,149.049
C02428=1162.072,31.506,-48.507,-179.829,6.112,149.049
C02429=1162.076,31.257,-48.492,-179.832,6.111,149.050
C02430=1162.081,31.008,-48.478,-179.834,6.110,149.050
C02431=1162.087,30.758,-48.462,-179.837,6.110,149.051
C02432=1162.092,30.508,-48.448,-179.839,6.108,149.052
C02433=1162.096,30.259,-48.433,-179.842,6.108,149.052
C02434=1162.101,30.010,-48.419,-179.844,6.107,149.053
C02435=1162.107,29.760,-48.403,-179.847,6.107,149.053
C02436=1162.111,29.510,-48.389,-179.850,6.105,149.054
C02437=1162.116,29.261,-48.374,-179.852,6.104,149.055
C02438=1162.122,29.011,-48.359,-179.855,6.104,149.055
C02439=1162.127,28.762,-48.345,-179.857,6.103,149.056
C02440=1162.131,28.513,-48.330,-179.860,6.102,149.056
C02441=1162.137,28.244,-48.314,-179.862,6.101,149.057
C02442=1162.142,27.975,-48.298,-179.865,6.101,149.057
C02443=1162.148,27.706,-48.282,-179.868,6.099,149.058
C02444=1162.153,27.436,-48.267,-179.870,6.098,149.059
C02445=1162.158,27.187,-48.251,-179.874,6.097,149.059
C02446=1162.163,26.937,-48.237,-179.876,6.097,149.060
C02447=1162.169,26.689,-48.222,-179.879,6.096,149.060
C02448=1162.174,26.439,-48.208,-179.881,6.095,149.061
C02449=1162.179,26.189,-48.193,-179.884,6.094,149.062
C02450=1162.184,25.940,-48.179,-179.887,6.093,149.062
C02451=1162.189,25.690,-48.164,-179.889,6.092,149.063
C02452=1162.194,25.441,-48.150,-179.891,6.092,149.063
C02453=1162.199,25.191,-48.135,-179.894,6.091,149.064
C02454=1162.204,24.942,-48.120,-179.897,6.090,149.064
C02455=1162.209,24.692,-48.105,-179.899,6.089,149.065
C02456=1162.214,24.442,-48.091,-179.902,6.088,149.066
C02457=1162.219,24.192,-48.077,-179.904,6.088,149.066
C02458=1162.224,23.944,-48.062,-179.907,6.086,149.067
C02459=1162.229,23.694,-48.048,-179.909,6.086,149.067
C02460=1162.234,23.445,-48.034,-179.912,6.085,149.068
C02461=1162.240,23.195,-48.019,-179.914,6.085,149.069
C02462=1162.245,22.945,-48.005,-179.917,6.084,149.069
C02463=1162.249,22.696,-47.990,-179.920,6.082,149.070
C02464=1162.254,22.446,-47.975,-179.922,6.082,149.070
C02465=1162.260,22.197,-47.961,-179.925,6.081,149.071
C02466=1162.265,21.947,-47.947,-179.927,6.080,149.071
C02467=1162.270,21.698,-47.933,-179.930,6.079,149.072
C02468=1162.275,21.449,-47.918,-179.932,6.078,149.072
C02469=1162.279,21.199,-47.904,-179.935,6.078,149.073
C02470=1162.284,20.949,-47.889,-179.937,6.077,149.074
C02471=1162.289,20.699,-47.875,-179.940,6.076,149.074
C02472=1162.296,20.450,-47.861,-179.942,6.075,149.075
C02473=1162.301,20.200,-47.846,-179.945,6.074,149.075
C02474=1162.306,19.951,-47.832,-179.948,6.074,149.076
C02475=1162.311,19.701,-47.818,-179.950,6.073,149.077
C02476=1162.315,19.451,-47.803,-179.953,6.073,149.077
C02477=1162.321,19.202,-47.790,-179.955,6.071,149.078
C02478=1162.326,18.953,-47.775,-179.958,6.070,149.078
C02479=1162.331,18.704,-47.760,-179.960,6.070,149.079
C02480=1162.336,18.454,-47.746,-179.963,6.069,149.079
C02481=1162.341,18.204,-47.732,-179.965,6.068,149.080
C02482=1162.346,17.955,-47.718,-179.968,6.068,149.081
C02483=1162.351,17.705,-47.703,-179.970,6.066,149.081
C02484=1162.356,17.456,-47.689,-179.973,6.066,149.082
C02485=1162.361,17.206,-47.675,-179.975,6.065,149.082
C02486=1162.367,16.957,-47.661,-179.978,6.064,149.083
C02487=1162.371,16.707,-47.647,-179.980,6.064,149.084
C02488=1162.376,16.458,-47.632,-179.983,6.062,149.084
C02489=1162.381,16.208,-47.618,-179.986,6.062,149.085
C02490=1162.386,15.958,-47.604,-179.988,6.061,149.085
C02491=1162.392,15.709,-47.590,-179.991,6.061,149.086
C02492=1162.396,15.459,-47.577,-179.993,6.060,149.086
C02493=1162.401,15.209,-47.563,-179.996,6.059,149.087
C02494=1162.407,14.960,-47.549,-179.998,6.058,149.087
C02495=1162.412,14.711,-47.535,179.999,6.057,149.088
C02496=1162.417,14.461,-47.520,179.996,6.057,149.089
C02497=1162.422,14.211,-47.506,179.994,6.056,149.089
C02498=1162.427,13.962,-47.492,179.992,6.055,149.090
C02499=1162.432,13.713,-47.478,179.989,6.055,149.090
C02500=1162.437,13.463,-47.464,179.986,6.053,149.091
C02501=1162.442,13.213,-47.449,179.984,6.052,149.092
C02502=1162.448,12.963,-47.436,179.981,6.052,149.092
C02503=1162.452,12.714,-47.422,179.979,6.051,149.093
C02504=1162.457,12.464,-47.408,179.977,6.051,149.093
C02505=1162.463,12.215,-47.394,179.974,6.050,149.094
C02506=1162.468,11.966,-47.380,179.971,6.049,149.095
C02507=1162.473,11.716,-47.366,179.968,6.048,149.095
C02508=1162.479,11.466,-47.352,179.966,6.047,149.096
C02509=1162.484,11.217,-47.338,179.964,6.047,149.096
C02510=1162.488,10.967,-47.325,179.961,6.046,149.097
C02511=1162.493,10.718,-47.311,179.959,6.046,149.097
C02512=1162.499,10.468,-47.297,179.957,6.045,149.098
C02513=1162.504,10.218,-47.283,179.953,6.043,149.099
C02514=1162.509,9.969,-47.269,179.951,6.043,149.099
C02515=1162.513,9.720,-47.255,179.949,6.042,149.100
C02516=1162.519,9.469,-47.242,179.946,6.042,149.100
C02517=1162.524,9.220,-47.228,179.944,6.041,149.101
C02518=1162.529,8.971,-47.213,179.941,6.040,149.102
C02519=1162.534,8.721,-47.199,179.939,6.040,149.102
C02520=1162.539,8.472,-47.187,179.936,6.039,149.103
C02521=1162.544,8.222,-47.172,179.934,6.038,149.103
C02522=1162.550,7.973,-47.158,179.931,6.037,149.104
C02523=1162.555,7.723,-47.145,179.929,6.036,149.104
C02524=1162.559,7.473,-47.131,179.926,6.036,149.105
C02525=1162.565,7.224,-47.117,179.923,6.035,149.106
C02526=1162.570,6.974,-47.104,179.921,6.034,149.106
C02527=1162.576,6.725,-47.090,179.919,6.034,149.107
C02528=1162.580,6.475,-47.076,179.916,6.033,149.107
C02529=1162.585,6.225,-47.062,179.913,6.032,149.108
C02530=1162.591,5.976,-47.049,179.911,6.031,149.108
C02531=1162.595,5.726,-47.036,179.908,6.031,149.109
C02532=1162.601,5.477,-47.022,179.906,6.030,149.110
C02533=1162.606,5.227,-47.007,179.904,6.029,149.110
C02534=1162.610,4.977,-46.994,179.901,6.029,149.111
C02535=1162.616,4.728,-46.981,179.899,6.028,149.111
C02536=1162.621,4.478,-46.967,179.896,6.028,149.112
C02537=1162.626,4.229,-46.954,179.894,6.027,149.113
C02538=1162.631,3.979,-46.940,179.891,6.026,149.113
C02539=1162.637,3.730,-46.926,179.888,6.025,149.114
C02540=1162.641,3.480,-46.913,179.886,6.024,149.114
C02541=1162.646,3.230,-46.899,179.884,6.023,149.115
C02542=1162.652,2.981,-46.886,179.881,6.023,149.116
C02543=1162.656,2.731,-46.872,179.878,6.023,149.116
C02544=1162.662,2.482,-46.859,179.876,6.022,149.117
C02545=1162.667,2.212,-46.844,179.873,6.021,149.117
C02546=1162.673,1.943,-46.829,179.870,6.020,149.118
C02547=1162.678,1.674,-46.815,179.868,6.019,149.119
C02548=1162.684,1.404,-46.801,179.865,6.019,149.119
C02549=1162.689,1.155,-46.786,179.863,6.018,149.120
C02550=1162.694,0.905,-46.774,179.861,6.017,149.120
C02551=1162.699,0.656,-46.759,179.858,6.017,149.121
C02552=1162.704,0.406,-46.747,179.856,6.016,149.122
C02553=1162.709,0.156,-46.733,179.853,6.015,149.122
C02554=1162.715,-0.093,-46.719,179.850,6.014,149.123
C02555=1162.719,-0.343,-46.706,179.848,6.014,149.123
C02556=1162.725,-0.592,-46.692,179.845,6.013,149.124
C02557=1162.729,-0.842,-46.679,179.843,6.012,149.125
C02558=1162.735,-1.092,-46.666,179.840,6.012,149.125
C02559=1162.740,-1.341,-46.653,179.838,6.011,149.126
C02560=1162.745,-1.591,-46.639,179.835,6.011,149.126
C02561=1162.751,-1.840,-46.627,179.833,6.010,149.127
C02562=1162.755,-2.090,-46.613,179.831,6.009,149.128
C02563=1162.761,-2.339,-46.600,179.828,6.009,149.128
C02564=1162.766,-2.589,-46.586,179.826,6.008,149.129
C02565=1162.771,-2.838,-46.573,179.823,6.008,149.129
C02566=1162.776,-3.088,-46.560,179.820,6.006,149.130
C02567=1162.781,-3.338,-46.547,179.818,6.006,149.131
C02568=1162.786,-3.588,-46.533,179.815,6.005,149.131
C02569=1162.791,-3.837,-46.520,179.813,6.004,149.132
C02570=1162.797,-4.086,-46.507,179.810,6.004,149.132
C02571=1162.802,-4.336,-46.494,179.808,6.003,149.133
C02572=1162.807,-4.585,-46.480,179.805,6.003,149.134
C02573=1162.812,-4.836,-46.467,179.803,6.002,149.134
C02574=1162.817,-5.085,-46.454,179.800,6.001,149.135
C02575=1162.822,-5.335,-46.441,179.798,6.000,149.135
C02576=1162.827,-5.584,-46.428,179.796,6.000,149.136
C02577=1162.833,-5.833,-46.414,179.793,6.000,149.137
C02578=1162.837,-6.084,-46.401,179.791,5.999,149.137
C02579=1162.843,-6.333,-46.388,179.788,5.998,149.138
C02580=1162.848,-6.583,-46.375,179.786,5.998,149.138
C02581=1162.853,-6.832,-46.361,179.783,5.997,149.139
C02582=1162.858,-7.081,-46.349,179.781,5.996,149.139
C02583=1162.863,-7.331,-46.336,179.779,5.996,149.140
C02584=1162.869,-7.581,-46.323,179.776,5.995,149.140
C02585=1162.874,-7.830,-46.310,179.774,5.995,149.141
C02586=1162.878,-8.080,-46.297,179.771,5.994,149.142
C02587=1162.884,-8.329,-46.283,179.769,5.993,149.142
C02588=1162.888,-8.579,-46.270,179.766,5.992,149.143
C02589=1162.894,-8.829,-46.257,179.763,5.991,149.143
C02590=1162.899,-9.078,-46.244,179.761,5.991,149.144
C02591=1162.904,-9.328,-46.231,179.759,5.990,149.145
C02592=1162.910,-9.578,-46.218,179.756,5.989,149.145
C02593=1162.915,-9.827,-46.206,179.753,5.989,149.146
C02594=1162.919,-10.077,-46.193,179.751,5.988,149.146
C02595=1162.925,-10.327,-46.179,179.748,5.988,149.147
C02596=1162.930,-10.576,-46.167,179.746,5.987,149.148
C02597=1162.935,-10.826,-46.154,179.744,5.987,149.148
C02598=1162.940,-11.075,-46.140,179.741,5.986,149.149
C02599=1162.946,-11.325,-46.127,179.739,5.985,149.150
C02600=1162.950,-11.575,-46.114,179.737,5.984,149.150
C02601=1162.955,-11.824,-46.102,179.734,5.984,149.151
C02602=1162.961,-12.074,-46.089,179.731,5.984,149.151
C02603=1162.966,-12.324,-46.076,179.729,5.983,149.152
C02604=1162.971,-12.573,-46.063,179.726,5.982,149.153
C02605=1162.976,-12.822,-46.050,179.724,5.981,149.153
C02606=1162.982,-13.072,-46.037,179.722,5.981,149.154
C02607=1162.986,-13.322,-46.024,179.719,5.980,149.154
C02608=1162.991,-13.571,-46.012,179.717,5.980,149.155
C02609=1162.997,-13.821,-46.000,179.714,5.979,149.156
C02610=1163.002,-14.072,-45.986,179.712,5.979,149.156
C02611=1163.007,-14.321,-45.974,179.709,5.978,149.157
C02612=1163.012,-14.570,-45.961,179.707,5.977,149.157
C02613=1163.017,-14.820,-45.948,179.704,5.977,149.158
C02614=1163.023,-15.070,-45.935,179.702,5.976,149.158
C02615=1163.028,-15.319,-45.922,179.700,5.976,149.159
C02616=1163.033,-15.568,-45.910,179.697,5.975,149.160
C02617=1163.038,-15.818,-45.897,179.695,5.974,149.160
C02618=1163.043,-16.068,-45.884,179.692,5.974,149.161
C02619=1163.048,-16.317,-45.871,179.690,5.973,149.161
C02620=1163.054,-16.567,-45.859,179.687,5.973,149.162
C02621=1163.059,-16.817,-45.846,179.685,5.972,149.162
C02622=1163.063,-17.067,-45.833,179.682,5.971,149.163
C02623=1163.069,-17.316,-45.821,179.680,5.971,149.164
C02624=1163.074,-17.565,-45.808,179.678,5.970,149.164
C02625=1163.079,-17.815,-45.796,179.675,5.970,149.165
C02626=1163.085,-18.065,-45.783,179.673,5.969,149.166
C02627=1163.090,-18.315,-45.770,179.670,5.968,149.166
C02628=1163.095,-18.564,-45.757,179.668,5.968,149.167
C02629=1163.100,-18.814,-45.745,179.665,5.967,149.167
C02630=1163.105,-19.063,-45.732,179.663,5.966,149.168
C02631=1163.110,-19.313,-45.720,179.660,5.966,149.169
C02632=1163.115,-19.563,-45.707,179.658,5.966,149.169
C02633=1163.121,-19.812,-45.694,179.656,5.965,149.170
C02634=1163.126,-20.062,-45.682,179.654,5.965,149.170
C02635=1163.131,-20.312,-45.670,179.651,5.964,149.171
C02636=1163.136,-20.561,-45.657,179.649,5.964,149.172
C02637=1163.141,-20.811,-45.644,179.647,5.963,149.172
C02638=1163.146,-21.060,-45.632,179.644,5.963,149.173
C02639=1163.151,-21.310,-45.620,179.641,5.962,149.173
C02640=1163.157,-21.560,-45.607,179.639,5.961,149.174
C02641=1163.162,-21.809,-45.595,179.636,5.961,149.175
C02642=1163.167,-22.059,-45.583,179.634,5.960,149.175
C02643=1163.172,-22.308,-45.570,179.632,5.960,149.176
C02644=1163.177,-22.558,-45.557,179.629,5.959,149.176
C02645=1163.182,-22.808,-45.545,179.627,5.958,149.177
C02646=1163.187,-23.057,-45.533,179.624,5.958,149.177
C02647=1163.192,-23.307,-45.520,179.622,5.957,149.178
C02648=1163.198,-23.557,-45.508,179.619,5.957,149.179
C02649=1163.204,-23.827,-45.494,179.617,5.956,149.179
C02650=1163.210,-24.096,-45.481,179.614,5.955,149.180
C02651=1163.215,-24.366,-45.468,179.612,5.955,149.181
C02652=1163.221,-24.637,-45.454,179.609,5.955,149.181
C02653=1163.226,-24.886,-45.441,179.607,5.954,149.182
C02654=1163.231,-25.136,-45.429,179.604,5.953,149.183
C02655=1163.236,-25.385,-45.417,179.602,5.953,149.183
C02656=1163.241,-25.635,-45.404,179.599,5.952,149.184
C02657=1163.247,-25.885,-45.392,179.597,5.951,149.184
C02658=1163.251,-26.134,-45.380,179.594,5.951,149.185
C02659=1163.257,-26.384,-45.368,179.592,5.950,149.186
C02660=1163.262,-26.633,-45.356,179.590,5.950,149.186
C02661=1163.267,-26.884,-45.344,179.587,5.949,149.187
C02662=1163.272,-27.133,-45.331,179.585,5.948,149.187
C02663=1163.277,-27.383,-45.319,179.582,5.948,149.188
C02664=1163.282,-27.632,-45.307,179.581,5.948,149.188
C02665=1163.288,-27.882,-45.295,179.578,5.948,149.189
C02666=1163.293,-28.131,-45.282,179.576,5.947,149.190
C02667=1163.298,-28.381,-45.270,179.573,5.946,149.190
C02668=1163.303,-28.631,-45.258,179.570,5.946,149.191
C02669=1163.309,-28.881,-45.246,179.568,5.945,149.191
C02670=1163.314,-29.130,-45.233,179.566,5.945,149.192
C02671=1163.319,-29.379,-45.222,179.563,5.944,149.193
C02672=1163.324,-29.629,-45.209,179.561,5.943,149.193
C02673=1163.329,-29.879,-45.197,179.559,5.943,149.194
C02674=1163.334,-30.128,-45.185,179.556,5.942,149.194
C02675=1163.340,-30.378,-45.173,179.553,5.942,149.195
C02676=1163.345,-30.628,-45.161,179.552,5.942,149.196
C02677=1163.350,-30.877,-45.148,179.549,5.941,149.196
C02678=1163.355,-31.127,-45.137,179.547,5.940,149.197
C02679=1163.360,-31.376,-45.124,179.544,5.940,149.197
C02680=1163.366,-31.626,-45.113,179.542,5.939,149.198
C02681=1163.371,-31.876,-45.101,179.539,5.939,149.199
C02682=1163.376,-32.125,-45.088,179.537,5.938,149.199
C02683=1163.382,-32.375,-45.076,179.534,5.938,149.200
C02684=1163.386,-32.625,-45.065,179.532,5.937,149.201
C02685=1163.391,-32.874,-45.052,179.530,5.936,149.201
C02686=1163.397,-33.124,-45.040,179.527,5.936,149.202
C02687=1163.402,-33.374,-45.029,179.525,5.936,149.202
C02688=1163.407,-33.623,-45.016,179.523,5.935,149.203
C02689=1163.412,-33.873,-45.005,179.520,5.935,149.203
C02690=1163.417,-34.123,-44.993,179.518,5.934,149.204
C02691=1163.423,-34.372,-44.980,179.516,5.933,149.204
C02692=1163.428,-34.622,-44.968,179.513,5.933,149.205
C02693=1163.433,-34.872,-44.956,179.510,5.933,149.206
C02694=1163.438,-35.121,-44.944,179.508,5.932,149.206
C02695=1163.443,-35.371,-44.933,179.505,5.931,149.207
C02696=1163.449,-35.621,-44.921,179.504,5.931,149.208
C02697=1163.454,-35.871,-44.909,179.501,5.931,149.208
C02698=1163.459,-36.120,-44.897,179.499,5.930,149.209
C02699=1163.464,-36.370,-44.885,179.496,5.930,149.209
C02700=1163.469,-36.620,-44.873,179.494,5.929,149.210
C02701=1163.474,-36.870,-44.862,179.491,5.928,149.211
C02702=1163.479,-37.119,-44.850,179.489,5.928,149.211
C02703=1163.485,-37.369,-44.837,179.487,5.927,149.212
C02704=1163.491,-37.618,-44.826,179.485,5.928,149.212
C02705=1163.495,-37.868,-44.814,179.482,5.927,149.213
C02706=1163.501,-38.118,-44.802,179.480,5.926,149.214
C02707=1163.506,-38.368,-44.791,179.478,5.926,149.214
C02708=1163.511,-38.617,-44.779,179.475,5.925,149.215
C02709=1163.516,-38.866,-44.767,179.473,5.924,149.215
C02710=1163.521,-39.116,-44.755,179.470,5.924,149.216
C02711=1163.526,-39.366,-44.744,179.468,5.923,149.216
C02712=1163.532,-39.616,-44.732,179.466,5.924,149.217
C02713=1163.538,-39.865,-44.720,179.463,5.923,149.218
C02714=1163.542,-40.115,-44.709,179.461,5.922,149.218
C02715=1163.548,-40.365,-44.697,179.458,5.922,149.219
C02716=1163.553,-40.614,-44.684,179.456,5.921,149.219
C02717=1163.558,-40.864,-44.673,179.453,5.921,149.220
C02718=1163.563,-41.114,-44.661,179.451,5.920,149.221
C02719=1163.568,-41.364,-44.649,179.449,5.920,149.221
C02720=1163.573,-41.613,-44.638,179.447,5.919,149.222
C02721=1163.579,-41.862,-44.626,179.444,5.919,149.223
C02722=1163.584,-42.112,-44.615,179.442,5.918,149.223
C02723=1163.589,-42.362,-44.603,179.439,5.918,149.224
C02724=1163.595,-42.612,-44.591,179.437,5.917,149.224
C02725=1163.599,-42.862,-44.580,179.435,5.917,149.225
C02726=1163.605,-43.112,-44.568,179.433,5.917,149.226
C02727=1163.610,-43.360,-44.557,179.430,5.916,149.226
C02728=1163.615,-43.610,-44.545,179.428,5.916,149.227
C02729=1163.621,-43.860,-44.534,179.426,5.915,149.227
C02730=1163.626,-44.110,-44.522,179.423,5.915,149.228
C02731=1163.631,-44.360,-44.510,179.421,5.914,149.228
C02732=1163.636,-44.609,-44.499,179.419,5.914,149.229
C02733=1163.642,-44.859,-44.488,179.416,5.913,149.230
C02734=1163.646,-45.108,-44.476,179.414,5.913,149.230
C02735=1163.652,-45.358,-44.464,179.412,5.912,149.231
C02736=1163.657,-45.608,-44.453,179.409,5.912,149.231
C02737=1163.662,-45.858,-44.441,179.406,5.911,149.232
C02738=1163.667,-46.107,-44.430,179.405,5.911,149.233
C02739=1163.673,-46.357,-44.418,179.402,5.911,149.233
C02740=1163.677,-46.606,-44.407,179.400,5.910,149.234
C02741=1163.683,-46.856,-44.395,179.397,5.910,149.235
C02742=1163.688,-47.106,-44.384,179.395,5.909,149.235
C02743=1163.694,-47.355,-44.372,179.392,5.908,149.236
C02744=1163.699,-47.605,-44.362,179.391,5.908,149.236
C02745=1163.704,-47.855,-44.350,179.388,5.908,149.237
C02746=1163.709,-48.105,-44.339,179.386,5.907,149.237
C02747=1163.715,-48.354,-44.327,179.383,5.907,149.238
C02748=1163.719,-48.604,-44.316,179.381,5.906,149.239
C02749=1163.725,-48.854,-44.304,179.379,5.906,149.239
C02750=1163.730,-49.103,-44.293,179.377,5.906,149.240
C02751=1163.736,-49.353,-44.282,179.374,5.905,149.240
C02752=1163.741,-49.603,-44.271,179.371,5.905,149.241
C02753=1163.746,-49.873,-44.258,179.369,5.904,149.242
C02754=1163.752,-50.143,-44.246,179.367,5.904,149.242
C02755=1163.758,-50.414,-44.234,179.364,5.903,149.243
C02756=1163.763,-50.685,-44.221,179.361,5.903,149.244
C02757=1163.769,-50.934,-44.210,179.359,5.902,149.244
C02758=1163.774,-51.184,-44.198,179.357,5.902,149.245
C02759=1163.779,-51.434,-44.187,179.355,5.902,149.245
C02760=1163.783,-51.684,-44.176,179.352,5.901,149.246
C02761=1163.790,-51.933,-44.165,179.350,5.900,149.247
C02762=1163.794,-52.183,-44.154,179.347,5.900,149.247
C02763=1163.799,-52.433,-44.142,179.346,5.900,149.248
C02764=1163.805,-52.682,-44.131,179.343,5.900,149.248
C02765=1163.810,-52.932,-44.120,179.341,5.899,149.249
C02766=1163.816,-53.182,-44.109,179.338,5.898,149.250
C02767=1163.821,-53.431,-44.098,179.336,5.898,149.250
C02768=1163.826,-53.681,-44.087,179.334,5.898,149.251
C02769=1163.831,-53.931,-44.075,179.332,5.897,149.251
C02770=1163.837,-54.180,-44.064,179.329,5.897,149.252
C02771=1163.841,-54.430,-44.053,179.327,5.896,149.252
C02772=1163.847,-54.680,-44.042,179.324,5.895,149.253
C02773=1163.852,-54.930,-44.030,179.323,5.895,149.254
C02774=1163.857,-55.179,-44.020,179.320,5.895,149.254
C02775=1163.863,-55.429,-44.008,179.318,5.894,149.255
C02776=1163.867,-55.679,-43.997,179.315,5.894,149.256
C02777=1163.873,-55.928,-43.986,179.313,5.894,149.256
C02778=1163.878,-56.178,-43.976,179.311,5.893,149.257
C02779=1163.884,-56.427,-43.964,179.308,5.893,149.257
C02780=1163.889,-56.678,-43.953,179.306,5.892,149.258
C02781=1163.893,-56.927,-43.942,179.303,5.892,149.259
C02782=1163.900,-57.177,-43.931,179.302,5.892,149.259
C02783=1163.904,-57.427,-43.920,179.299,5.891,149.260
C02784=1163.909,-57.676,-43.909,179.297,5.891,149.260
C02785=1163.915,-57.926,-43.899,179.294,5.890,149.261
C02786=1163.920,-58.176,-43.887,179.293,5.890,149.261
C02787=1163.925,-58.425,-43.875,179.290,5.890,149.262
C02788=1163.931,-58.675,-43.865,179.288,5.889,149.263
C02789=1163.935,-58.925,-43.854,179.285,5.889,149.263
C02790=1163.942,-59.175,-43.843,179.283,5.888,149.264
C02791=1163.946,-59.424,-43.832,179.281,5.888,149.265
C02792=1163.951,-59.674,-43.821,179.279,5.887,149.265
C02793=1163.957,-59.923,-43.810,179.276,5.887,149.266
C02794=1163.962,-60.174,-43.800,179.274,5.886,149.266
C02795=1163.968,-60.423,-43.788,179.272,5.887,149.267
C02796=1163.973,-60.673,-43.778,179.269,5.886,149.267
C02797=1163.977,-60.923,-43.766,179.267,5.885,149.268
C02798=1163.983,-61.172,-43.756,179.265,5.885,149.269
C02799=1163.988,-61.422,-43.745,179.263,5.885,149.269
C02800=1163.994,-61.672,-43.734,179.260,5.884,149.270
C02801=1163.999,-61.921,-43.723,179.258,5.884,149.270
C02802=1164.004,-62.171,-43.713,179.255,5.883,149.271
C02803=1164.009,-62.420,-43.701,179.253,5.883,149.272
C02804=1164.014,-62.671,-43.691,179.251,5.883,149.272
C02805=1164.019,-62.920,-43.680,179.249,5.882,149.273
C02806=1164.025,-63.170,-43.669,179.246,5.882,149.273
C02807=1164.030,-63.420,-43.658,179.244,5.882,149.274
C02808=1164.035,-63.669,-43.647,179.242,5.881,149.274
C02809=1164.041,-63.919,-43.637,179.239,5.881,149.275
C02810=1164.045,-64.169,-43.626,179.237,5.880,149.276
C02811=1164.051,-64.418,-43.615,179.235,5.880,149.276
C02812=1164.056,-64.668,-43.605,179.233,5.880,149.277
C02813=1164.062,-64.918,-43.593,179.230,5.879,149.278
C02814=1164.067,-65.168,-43.583,179.228,5.878,149.278
C02815=1164.072,-65.417,-43.572,179.226,5.879,149.279
C02816=1164.077,-65.667,-43.561,179.224,5.878,149.279
C02817=1164.082,-65.917,-43.551,179.221,5.878,149.280
C02818=1164.088,-66.166,-43.540,179.219,5.877,149.280
C02819=1164.093,-66.416,-43.529,179.217,5.877,149.281
C02820=1164.098,-66.666,-43.519,179.215,5.876,149.282
C02821=1164.103,-66.916,-43.508,179.212,5.876,149.282
C02822=1164.109,-67.165,-43.497,179.211,5.876,149.283
C02823=1164.114,-67.415,-43.487,179.208,5.876,149.283
C02824=1164.120,-67.665,-43.475,179.206,5.875,149.284
C02825=1164.125,-67.914,-43.465,179.203,5.874,149.285
C02826=1164.130,-68.164,-43.455,179.201,5.874,149.285
C02827=1164.136,-68.414,-43.444,179.199,5.874,149.286
C02828=1164.140,-68.664,-43.433,179.197,5.873,149.286
C02829=1164.146,-68.913,-43.423,179.194,5.873,149.287
C02830=1164.151,-69.163,-43.412,179.192,5.873,149.288
C02831=1164.157,-69.413,-43.402,179.190,5.872,149.288
C02832=1164.161,-69.662,-43.391,179.187,5.872,149.289
C02833=1164.167,-69.912,-43.381,179.185,5.872,149.289
C02834=1164.172,-70.162,-43.370,179.183,5.871,149.290
C02835=1164.178,-70.412,-43.360,179.180,5.871,149.291
C02836=1164.182,-70.661,-43.349,179.178,5.870,149.291
C02837=1164.188,-70.911,-43.338,179.176,5.870,149.292
C02838=1164.193,-71.161,-43.328,179.174,5.870,149.292
C02839=1164.198,-71.411,-43.318,179.171,5.869,149.293
C02840=1164.204,-71.660,-43.307,179.170,5.869,149.293
C02841=1164.209,-71.910,-43.296,179.167,5.869,149.294
C02842=1164.214,-72.159,-43.286,179.165,5.868,149.295
C02843=1164.219,-72.410,-43.275,179.163,5.867,149.295
C02844=1164.225,-72.659,-43.265,179.161,5.868,149.296
C02845=1164.231,-72.909,-43.255,179.158,5.867,149.296
C02846=1164.236,-73.159,-43.244,179.156,5.867,149.297
C02847=1164.241,-73.409,-43.234,179.154,5.867,149.297
C02848=1164.246,-73.658,-43.223,179.151,5.866,149.298
C02849=1164.251,-73.908,-43.213,179.149,5.865,149.299
C02850=1164.257,-74.157,-43.202,179.147,5.866,149.299
C02851=1164.261,-74.407,-43.192,179.145,5.865,149.300
C02852=1164.267,-74.657,-43.182,179.142,5.865,149.301
C02853=1164.272,-74.906,-43.172,179.140,5.864,149.301
C02854=1164.277,-75.157,-43.161,179.138,5.864,149.302
C02855=1164.283,-75.406,-43.151,179.136,5.863,149.302
C02856=1164.288,-75.656,-43.141,179.133,5.863,149.303
C02857=1164.295,-75.927,-43.129,179.132,5.863,149.303
C02858=1164.299,-76.198,-43.118,179.129,5.863,149.304
C02859=1164.305,-76.470,-43.106,179.126,5.862,149.305
C02860=1164.311,-76.740,-43.096,179.124,5.861,149.305
C02861=1164.316,-76.990,-43.085,179.121,5.861,149.306
C02862=1164.322,-77.240,-43.075,179.120,5.861,149.307
C02863=1164.327,-77.489,-43.065,179.117,5.861,149.307
C02864=1164.332,-77.740,-43.054,179.115,5.860,149.308
C02865=1164.338,-77.989,-43.044,179.113,5.860,149.308
C02866=1164.343,-78.239,-43.034,179.111,5.860,149.309
C02867=1164.348,-78.489,-43.024,179.108,5.859,149.310
C02868=1164.353,-78.738,-43.013,179.106,5.859,149.310
C02869=1164.359,-78.988,-43.003,179.104,5.859,149.311
C02870=1164.364,-79.238,-42.993,179.102,5.858,149.311
C02871=1164.370,-79.488,-42.982,179.100,5.858,149.312
C02872=1164.374,-79.737,-42.973,179.097,5.858,149.312
C02873=1164.379,-79.987,-42.962,179.095,5.857,149.313
C02874=1164.385,-80.237,-42.952,179.093,5.857,149.314
C02875=1164.391,-80.486,-42.942,179.091,5.856,149.314
C02876=1164.396,-80.737,-42.932,179.088,5.856,149.315
C02877=1164.401,-80.986,-42.922,179.087,5.856,149.315
C02878=1164.406,-81.236,-42.912,179.084,5.856,149.316
C02879=1164.412,-81.485,-42.902,179.082,5.855,149.317
C02880=1164.417,-81.736,-42.891,179.080,5.855,149.317
C02881=1164.423,-81.985,-42.881,179.077,5.855,149.318
C02882=1164.427,-82.234,-42.872,179.075,5.854,149.318
C02883=1164.432,-82.485,-42.861,179.073,5.854,149.319
C02884=1164.438,-82.734,-42.851,179.071,5.853,149.319
C02885=1164.444,-82.984,-42.841,179.068,5.853,149.320
C02886=1164.449,-83.234,-42.832,179.067,5.853,149.321
C02887=1164.454,-83.484,-42.821,179.064,5.853,149.321
C02888=1164.459,-83.733,-42.811,179.062,5.852,149.322
C02889=1164.465,-83.983,-42.801,179.060,5.852,149.322
C02890=1164.470,-84.232,-42.791,179.058,5.851,149.323
C02891=1164.475,-84.482,-42.781,179.055,5.851,149.323
C02892=1164.481,-84.733,-42.771,179.053,5.851,149.324
C02893=1164.486,-84.982,-42.761,179.051,5.850,149.325
C02894=1164.491,-85.231,-42.751,179.048,5.850,149.325
C02895=1164.496,-85.482,-42.741,179.047,5.850,149.326
C02896=1164.501,-85.731,-42.731,179.044,5.850,149.327
C02897=1164.507,-85.981,-42.722,179.042,5.849,149.327
C02898=1164.513,-86.231,-42.711,179.040,5.849,149.328
C02899=1164.518,-86.481,-42.701,179.038,5.848,149.328
C02900=1164.522,-86.730,-42.691,179.036,5.848,149.329
C02901=1164.528,-86.980,-42.681,179.033,5.848,149.329
C02902=1164.534,-87.230,-42.671,179.031,5.847,149.330
C02903=1164.538,-87.480,-42.661,179.029,5.848,149.331
C02904=1164.544,-87.729,-42.651,179.027,5.847,149.331
C02905=1164.549,-87.979,-42.642,179.025,5.846,149.332
C02906=1164.555,-88.229,-42.632,179.023,5.847,149.332
C02907=1164.560,-88.478,-42.622,179.021,5.846,149.333
C02908=1164.564,-88.728,-42.612,179.018,5.845,149.334
C02909=1164.570,-88.978,-42.602,179.016,5.845,149.334
C02910=1164.576,-89.228,-42.592,179.014,5.845,149.335
C02911=1164.581,-89.477,-42.583,179.011,5.844,149.335
C02912=1164.587,-89.727,-42.573,179.010,5.844,149.336
C02913=1164.591,-89.977,-42.563,179.007,5.844,149.336
C02914=1164.597,-90.227,-42.553,179.006,5.844,149.337
C02915=1164.602,-90.477,-42.543,179.003,5.843,149.338
C02916=1164.607,-90.726,-42.534,179.001,5.843,149.338
C02917=1164.613,-90.976,-42.524,178.999,5.843,149.339
C02918=1164.618,-91.225,-42.515,178.996,5.842,149.339
C02919=1164.623,-91.476,-42.504,178.994,5.842,149.340
C02920=1164.629,-91.725,-42.494,178.992,5.842,149.340
C02921=1164.634,-91.975,-42.485,178.990,5.841,149.341
C02922=1164.639,-92.225,-42.475,178.988,5.842,149.342
C02923=1164.645,-92.474,-42.466,178.986,5.841,149.342
C02924=1164.650,-92.724,-42.456,178.983,5.840,149.343
C02925=1164.655,-92.973,-42.446,178.981,5.840,149.343
C02926=1164.660,-93.224,-42.436,178.979,5.840,149.344
C02927=1164.666,-93.474,-42.426,178.977,5.840,149.345
C02928=1164.671,-93.723,-42.417,178.975,5.839,149.345
C02929=1164.677,-93.973,-42.407,178.973,5.839,149.345
C02930=1164.682,-94.222,-42.397,178.971,5.839,149.346
C02931=1164.688,-94.472,-42.388,178.968,5.838,149.347
C02932=1164.692,-94.722,-42.378,178.966,5.838,149.347
C02933=1164.698,-94.973,-42.368,178.964,5.838,149.348
C02934=1164.703,-95.222,-42.359,178.962,5.837,149.348
C02935=1164.708,-95.472,-42.349,178.960,5.837,149.349
C02936=1164.713,-95.721,-42.340,178.958,5.837,149.350
C02937=1164.719,-95.971,-42.330,178.955,5.836,149.350
C02938=1164.724,-96.221,-42.321,178.953,5.836,149.351
C02939=1164.730,-96.471,-42.311,178.951,5.836,149.351
C02940=1164.735,-96.720,-42.301,178.949,5.836,149.352
C02941=1164.741,-96.970,-42.292,178.947,5.835,149.352
C02942=1164.746,-97.219,-42.282,178.944,5.835,149.353
C02943=1164.752,-97.469,-42.273,178.943,5.835,149.354
C02944=1164.756,-97.719,-42.263,178.941,5.834,149.354
C02945=1164.762,-97.970,-42.253,178.938,5.835,149.355
C02946=1164.767,-98.219,-42.244,178.936,5.834,149.355
C02947=1164.772,-98.469,-42.235,178.934,5.833,149.356
C02948=1164.778,-98.719,-42.225,178.932,5.833,149.356
C02949=1164.782,-98.968,-42.216,178.930,5.833,149.357
C02950=1164.788,-99.218,-42.206,178.928,5.833,149.358
C02951=1164.793,-99.467,-42.197,178.926,5.832,149.358
C02952=1164.799,-99.718,-42.187,178.923,5.831,149.359
C02953=1164.804,-99.967,-42.178,178.921,5.832,149.359
C02954=1164.810,-100.217,-42.168,178.919,5.831,149.360
C02955=1164.815,-100.467,-42.159,178.917,5.832,149.361
C02956=1164.820,-100.716,-42.150,178.915,5.831,149.361
C02957=1164.826,-100.966,-42.140,178.913,5.831,149.362
C02958=1164.831,-101.215,-42.130,178.911,5.830,149.362
C02959=1164.836,-101.465,-42.122,178.908,5.830,149.363
C02960=1164.842,-101.715,-42.112,178.907,5.830,149.363
C02961=1164.847,-101.987,-42.102,178.904,5.829,149.364
C02962=1164.853,-102.259,-42.092,178.901,5.829,149.365
C02963=1164.858,-102.531,-42.081,178.900,5.829,149.365
C02964=1164.864,-102.804,-42.071,178.897,5.829,149.366
C02965=1164.870,-103.053,-42.062,178.895,5.828,149.366
C02966=1164.874,-103.303,-42.052,178.893,5.828,149.367
C02967=1164.880,-103.553,-42.043,178.891,5.827,149.368
C02968=1164.886,-103.803,-42.034,178.889,5.827,149.368
C02969=1164.891,-104.052,-42.025,178.886,5.827,149.369
C02970=1164.896,-104.302,-42.015,178.884,5.826,149.369
C02971=1164.901,-104.552,-42.006,178.883,5.826,149.370
C02972=1164.907,-104.802,-41.997,178.880,5.826,149.370
C02973=1164.912,-105.051,-41.987,178.878,5.826,149.371
C02974=1164.917,-105.301,-41.978,178.876,5.825,149.371
C02975=1164.923,-105.551,-41.969,178.874,5.826,149.372
C02976=1164.929,-105.800,-41.960,178.872,5.825,149.373
C02977=1164.934,-106.050,-41.950,178.870,5.824,149.373
C02978=1164.939,-106.299,-41.941,178.868,5.825,149.374
C02979=1164.944,-106.549,-41.932,178.865,5.824,149.374
C02980=1164.950,-106.799,-41.923,178.864,5.824,149.375
C02981=1164.955,-107.049,-41.913,178.861,5.823,149.375
C02982=1164.960,-107.299,-41.904,178.860,5.823,149.376
C02983=1164.966,-107.549,-41.895,178.857,5.823,149.377
C02984=1164.971,-107.799,-41.886,178.855,5.823,149.377
C02985=1164.976,-108.048,-41.877,178.853,5.822,149.378
C02986=1164.981,-108.298,-41.867,178.850,5.822,149.378
C02987=1164.987,-108.548,-41.858,178.849,5.822,149.379
C02988=1164.992,-108.798,-41.849,178.847,5.821,149.379
C02989=1164.998,-109.048,-41.840,178.844,5.822,149.380
C02990=1165.003,-109.297,-41.831,178.842,5.821,149.381
C02991=1165.009,-109.548,-41.822,178.841,5.821,149.381
C02992=1165.013,-109.797,-41.812,178.838,5.821,149.382
C02993=1165.019,-110.047,-41.803,178.836,5.821,149.382
C02994=1165.024,-110.296,-41.795,178.834,5.820,149.383
C02995=1165.030,-110.546,-41.786,178.832,5.819,149.383
C02996=1165.035,-110.796,-41.776,178.830,5.819,149.384
C02997=1165.041,-111.046,-41.767,178.828,5.819,149.384
C02998=1165.046,-111.296,-41.758,178.826,5.819,149.385
C02999=1165.051,-111.545,-41.749,178.823,5.818,149.386
C03000=1165.057,-111.795,-41.739,178.822,5.818,149.386
C03001=1165.062,-112.045,-41.730,178.819,5.818,149.387
C03002=1165.067,-112.295,-41.721,178.818,5.818,149.387
C03003=1165.072,-112.544,-41.713,178.815,5.817,149.388
C03004=1165.078,-112.794,-41.704,178.813,5.818,149.388
C03005=1165.083,-113.043,-41.695,178.811,5.817,149.389
C03006=1165.089,-113.294,-41.686,178.810,5.817,149.389
C03007=1165.094,-113.543,-41.677,178.807,5.816,149.390
C03008=1165.099,-113.793,-41.668,178.805,5.816,149.391
C03009=1165.104,-114.043,-41.659,178.803,5.816,149.391
C03010=1165.110,-114.293,-41.650,178.801,5.815,149.392
C03011=1165.115,-114.543,-41.641,178.799,5.816,149.392
C03012=1165.121,-114.792,-41.632,178.797,5.815,149.393
C03013=1165.126,-115.042,-41.623,178.795,5.815,149.393
C03014=1165.132,-115.292,-41.614,178.792,5.814,149.394
C03015=1165.137,-115.542,-41.605,178.791,5.814,149.395
C03016=1165.142,-115.792,-41.596,178.789,5.814,149.395
C03017=1165.147,-116.042,-41.588,178.786,5.814,149.396
C03018=1165.153,-116.291,-41.579,178.784,5.813,149.396
C03019=1165.158,-116.541,-41.570,178.783,5.813,149.397
C03020=1165.164,-116.791,-41.561,178.780,5.813,149.397
C03021=1165.169,-117.041,-41.552,178.778,5.813,149.398
C03022=1165.174,-117.290,-41.543,178.776,5.812,149.398
C03023=1165.179,-117.540,-41.534,178.775,5.812,149.399
C03024=1165.185,-117.789,-41.525,178.772,5.812,149.400
C03025=1165.190,-118.039,-41.516,178.770,5.811,149.400
C03026=1165.196,-118.289,-41.508,178.768,5.811,149.401
C03027=1165.201,-118.539,-41.499,178.765,5.811,149.401
C03028=1165.206,-118.789,-41.490,178.764,5.811,149.402
C03029=1165.212,-119.038,-41.481,178.762,5.810,149.402
C03030=1165.217,-119.288,-41.473,178.760,5.810,149.403
C03031=1165.222,-119.538,-41.464,178.757,5.810,149.403
C03032=1165.227,-119.788,-41.455,178.756,5.810,149.404
C03033=1165.233,-120.038,-41.446,178.754,5.809,149.404
C03034=1165.238,-120.287,-41.438,178.752,5.809,149.405
C03035=1165.244,-120.537,-41.429,178.749,5.809,149.406
C03036=1165.249,-120.787,-41.420,178.748,5.809,149.406
C03037=1165.254,-121.037,-41.411,178.746,5.808,149.407
C03038=1165.260,-121.287,-41.402,178.743,5.808,149.407
C03039=1165.266,-121.537,-41.394,178.741,5.808,149.408
C03040=1165.271,-121.787,-41.385,178.740,5.808,149.408
C03041=1165.276,-122.036,-41.376,178.737,5.807,149.409
C03042=1165.281,-122.286,-41.367,178.735,5.807,149.409
C03043=1165.287,-122.535,-41.359,178.733,5.807,149.410
C03044=1165.292,-122.785,-41.350,178.732,5.807,149.410
C03045=1165.297,-123.035,-41.342,178.729,5.806,149.411
C03046=1165.302,-123.285,-41.333,178.727,5.806,149.412
C03047=1165.308,-123.534,-41.325,178.725,5.806,149.412
C03048=1165.313,-123.784,-41.316,178.724,5.806,149.413
C03049=1165.318,-124.034,-41.307,178.721,5.805,149.413
C03050=1165.324,-124.285,-41.299,178.719,5.805,149.414
C03051=1165.330,-124.534,-41.290,178.717,5.804,149.414
C03052=1165.335,-124.784,-41.281,178.715,5.804,149.415
C03053=1165.340,-125.033,-41.272,178.713,5.804,149.416
C03054=1165.345,-125.284,-41.264,178.711,5.804,149.416
C03055=1165.351,-125.533,-41.256,178.709,5.803,149.417
C03056=1165.356,-125.783,-41.247,178.707,5.803,149.417
C03057=1165.361,-126.033,-41.238,178.705,5.803,149.418
C03058=1165.367,-126.283,-41.230,178.703,5.803,149.418
C03059=1165.373,-126.532,-41.221,178.701,5.802,149.419
C03060=1165.378,-126.782,-41.212,178.699,5.802,149.419
C03061=1165.383,-127.033,-41.204,178.697,5.802,149.420
C03062=1165.389,-127.282,-41.196,178.695,5.802,149.420
C03063=1165.394,-127.531,-41.187,178.693,5.801,149.421
C03064=1165.399,-127.781,-41.178,178.691,5.801,149.421
C03065=1164.978,-127.792,-41.219,178.687,5.805,149.423
C03066=1164.973,-127.543,-41.228,178.690,5.805,149.423
C03067=1164.968,-127.293,-41.237,178.691,5.805,149.422
C03068=1164.962,-127.044,-41.246,178.693,5.806,149.422
C03069=1164.956,-126.793,-41.254,178.695,5.806,149.421
C03070=1164.951,-126.543,-41.263,178.698,5.806,149.421
C03071=1164.945,-126.294,-41.271,178.699,5.806,149.420
C03072=1164.941,-126.044,-41.279,178.701,5.807,149.420
C03073=1164.935,-125.794,-41.288,178.703,5.807,149.419
C03074=1164.930,-125.544,-41.297,178.706,5.807,149.418
C03075=1164.925,-125.295,-41.305,178.707,5.807,149.418
C03076=1164.919,-125.045,-41.314,178.709,5.808,149.417
C03077=1164.914,-124.795,-41.322,178.712,5.808,149.417
C03078=1164.909,-124.545,-41.331,178.714,5.808,149.416
C03079=1164.903,-124.296,-41.340,178.715,5.808,149.416
C03080=1164.897,-124.045,-41.348,178.718,5.809,149.415
C03081=1164.892,-123.795,-41.357,178.720,5.809,149.414
C03082=1164.887,-123.546,-41.365,178.722,5.810,149.414
C03083=1164.881,-123.296,-41.374,178.723,5.810,149.413
C03084=1164.876,-123.047,-41.383,178.726,5.810,149.413
C03085=1164.871,-122.796,-41.391,178.728,5.810,149.412
C03086=1164.865,-122.547,-41.400,178.730,5.811,149.412
C03087=1164.860,-122.297,-41.409,178.731,5.811,149.411
C03088=1164.855,-122.047,-41.418,178.734,5.811,149.411
C03089=1164.849,-121.797,-41.427,178.736,5.811,149.410
C03090=1164.844,-121.548,-41.436,178.738,5.812,149.410
C03091=1164.838,-121.298,-41.443,178.740,5.812,149.409
C03092=1164.833,-121.048,-41.452,178.742,5.812,149.408
C03093=1164.828,-120.798,-41.461,178.744,5.812,149.408
C03094=1164.823,-120.548,-41.470,178.746,5.813,149.407
C03095=1164.817,-120.299,-41.479,178.748,5.813,149.407
C03096=1164.812,-120.049,-41.488,178.750,5.813,149.406
C03097=1164.807,-119.799,-41.496,178.752,5.813,149.406
C03098=1164.801,-119.549,-41.505,178.754,5.814,149.405
C03099=1164.796,-119.299,-41.513,178.756,5.813,149.405
C03100=1164.790,-119.050,-41.522,178.758,5.814,149.404
C03101=1164.785,-118.800,-41.531,178.760,5.814,149.404
C03102=1164.780,-118.550,-41.540,178.762,5.815,149.403
C03103=1164.775,-118.300,-41.549,178.764,5.814,149.402
C03104=1164.770,-118.051,-41.558,178.766,5.815,149.402
C03105=1164.764,-117.801,-41.566,178.768,5.815,149.401
C03106=1164.758,-117.551,-41.576,178.771,5.816,149.401
C03107=1164.753,-117.301,-41.585,178.772,5.815,149.400
C03108=1164.748,-117.051,-41.593,178.775,5.816,149.400
C03109=1164.742,-116.802,-41.602,178.776,5.816,149.399
C03110=1164.737,-116.552,-41.611,178.779,5.817,149.399
C03111=1164.731,-116.303,-41.620,178.780,5.817,149.398
C03112=1164.726,-116.053,-41.629,178.783,5.817,149.398
C03113=1164.721,-115.803,-41.638,178.785,5.818,149.397
C03114=1164.716,-115.553,-41.646,178.787,5.818,149.396
C03115=1164.711,-115.303,-41.655,178.789,5.818,149.396
C03116=1164.705,-115.053,-41.665,178.791,5.818,149.395
C03117=1164.699,-114.804,-41.673,178.793,5.819,149.395
C03118=1164.694,-114.554,-41.682,178.795,5.819,149.394
C03119=1164.689,-114.304,-41.691,178.797,5.820,149.394
C03120=1164.684,-114.054,-41.700,178.799,5.819,149.393
C03121=1164.678,-113.805,-41.709,178.801,5.820,149.392
C03122=1164.673,-113.554,-41.718,178.803,5.820,149.392
C03123=1164.667,-113.304,-41.727,178.806,5.820,149.391
C03124=1164.662,-113.055,-41.736,178.807,5.820,149.391
C03125=1164.656,-112.806,-41.745,178.809,5.821,149.390
C03126=1164.651,-112.556,-41.754,178.812,5.820,149.390
C03127=1164.646,-112.306,-41.763,178.814,5.821,149.389
C03128=1164.640,-112.056,-41.772,178.816,5.822,149.389
C03129=1164.635,-111.806,-41.781,178.818,5.822,149.388
C03130=1164.630,-111.556,-41.790,178.820,5.822,149.387
C03131=1164.625,-111.306,-41.799,178.822,5.822,149.387
C03132=1164.620,-111.056,-41.808,178.824,5.823,149.386
C03133=1164.614,-110.807,-41.818,178.826,5.823,149.386
C03134=1164.608,-110.558,-41.826,178.828,5.823,149.385
C03135=1164.603,-110.308,-41.835,178.830,5.823,149.385
C03136=1164.598,-110.058,-41.844,178.833,5.824,149.384
C03137=1164.593,-109.808,-41.853,178.834,5.824,149.384
C03138=1164.587,-109.558,-41.863,178.837,5.824,149.383
C03139=1164.582,-109.308,-41.872,178.839,5.825,149.382
C03140=1164.577,-109.059,-41.881,178.841,5.825,149.382
C03141=1164.572,-108.809,-41.890,178.843,5.825,149.381
C03142=1164.566,-108.559,-41.900,178.845,5.825,149.381
C03143=1164.561,-108.309,-41.908,178.847,5.826,149.380
C03144=1164.555,-108.059,-41.917,178.849,5.826,149.379
C03145=1164.550,-107.809,-41.926,178.851,5.826,149.379
C03146=1164.545,-107.560,-41.936,178.853,5.826,149.379
C03147=1164.539,-107.310,-41.945,178.856,5.827,149.378
C03148=1164.534,-107.061,-41.954,178.858,5.827,149.377
C03149=1164.528,-106.811,-41.963,178.859,5.827,149.377
C03150=1164.523,-106.561,-41.972,178.862,5.828,149.376
C03151=1164.518,-106.311,-41.982,178.864,5.828,149.376
C03152=1164.513,-106.062,-41.991,178.866,5.829,149.375
C03153=1164.507,-105.811,-42.000,178.868,5.828,149.374
C03154=1164.501,-105.562,-42.009,178.870,5.829,149.374
C03155=1164.497,-105.312,-42.019,178.872,5.830,149.373
C03156=1164.491,-105.062,-42.028,178.874,5.829,149.373
C03157=1164.486,-104.812,-42.037,178.877,5.830,149.372
C03158=1164.480,-104.562,-42.046,178.878,5.830,149.372
C03159=1164.476,-104.313,-42.056,178.881,5.830,149.371
C03160=1164.470,-104.063,-42.065,178.882,5.830,149.371
C03161=1164.464,-103.813,-42.074,178.885,5.831,149.370
C03162=1164.460,-103.564,-42.084,178.887,5.831,149.369
C03163=1164.454,-103.314,-42.093,178.889,5.831,149.369
C03164=1164.449,-103.064,-42.102,178.892,5.832,149.368
C03165=1164.444,-102.815,-42.112,178.893,5.832,149.368
C03166=1164.437,-102.542,-42.122,178.896,5.832,149.367
C03167=1164.432,-102.270,-42.132,178.898,5.833,149.366
C03168=1164.426,-101.998,-42.142,178.900,5.833,149.366
C03169=1164.420,-101.727,-42.152,178.902,5.833,149.365
C03170=1164.414,-101.477,-42.162,178.905,5.834,149.365
C03171=1164.409,-101.227,-42.171,178.907,5.834,149.364
C03172=1164.405,-100.977,-42.180,178.909,5.834,149.364
C03173=1164.399,-100.727,-42.191,178.911,5.834,149.363
C03174=1164.394,-100.477,-42.200,178.913,5.835,149.362
C03175=1164.388,-100.227,-42.209,178.915,5.836,149.362
C03176=1164.383,-99.978,-42.219,178.917,5.835,149.361
C03177=1164.378,-99.728,-42.228,178.920,5.836,149.361
C03178=1164.372,-99.479,-42.238,178.922,5.835,149.360
C03179=1164.367,-99.229,-42.247,178.924,5.836,149.360
C03180=1164.362,-98.979,-42.257,178.926,5.837,149.359
C03181=1164.356,-98.729,-42.266,178.928,5.837,149.358
C03182=1164.351,-98.479,-42.275,178.930,5.837,149.358
C03183=1164.346,-98.230,-42.285,178.932,5.837,149.357
C03184=1164.341,-97.980,-42.294,178.935,5.838,149.357
C03185=1164.335,-97.731,-42.304,178.937,5.838,149.356
C03186=1164.330,-97.481,-42.313,178.939,5.838,149.355
C03187=1164.324,-97.231,-42.323,178.941,5.839,149.355
C03188=1164.319,-96.981,-42.332,178.943,5.839,149.354
C03189=1164.313,-96.732,-42.342,178.945,5.839,149.354
C03190=1164.309,-96.481,-42.351,178.948,5.840,149.353
C03191=1164.303,-96.232,-42.362,178.950,5.840,149.353
C03192=1164.298,-95.982,-42.371,178.952,5.840,149.352
C03193=1164.292,-95.732,-42.381,178.953,5.840,149.352
C03194=1164.287,-95.482,-42.390,178.956,5.841,149.351
C03195=1164.282,-95.233,-42.400,178.958,5.841,149.350
C03196=1164.277,-94.983,-42.409,178.960,5.841,149.350
C03197=1164.271,-94.734,-42.419,178.963,5.842,149.349
C03198=1164.266,-94.484,-42.428,178.964,5.842,149.349
C03199=1164.261,-94.233,-42.438,178.967,5.842,149.348
C03200=1164.256,-93.984,-42.447,178.969,5.843,149.348
C03201=1164.250,-93.734,-42.458,178.971,5.843,149.347
C03202=1164.245,-93.484,-42.466,178.973,5.843,149.346
C03203=1164.239,-93.235,-42.477,178.975,5.844,149.346
C03204=1164.234,-92.985,-42.487,178.978,5.844,149.345
C03205=1164.229,-92.735,-42.496,178.980,5.844,149.345
C03206=1164.223,-92.486,-42.506,178.982,5.844,149.344
C03207=1164.218,-92.235,-42.515,178.984,5.845,149.343
C03208=1164.213,-91.986,-42.525,178.986,5.846,149.343
C03209=1164.208,-91.736,-42.535,178.988,5.845,149.342
C03210=1164.202,-91.486,-42.545,178.990,5.846,149.342
C03211=1164.196,-91.237,-42.555,178.993,5.846,149.341
C03212=1164.192,-90.987,-42.564,178.995,5.846,149.341
C03213=1164.186,-90.737,-42.574,178.997,5.847,149.340
C03214=1164.181,-90.487,-42.584,178.999,5.847,149.339
C03215=1164.175,-90.237,-42.593,179.001,5.847,149.339
C03216=1164.171,-89.988,-42.603,179.004,5.848,149.338
C03217=1164.165,-89.738,-42.613,179.005,5.848,149.338
C03218=1164.159,-89.489,-42.623,179.008,5.849,149.337
C03219=1164.155,-89.238,-42.633,179.010,5.849,149.337
C03220=1164.149,-88.989,-42.643,179.012,5.849,149.336
C03221=1164.144,-88.739,-42.653,179.015,5.849,149.335
C03222=1164.138,-88.489,-42.662,179.016,5.849,149.335
C03223=1164.133,-88.240,-42.672,179.019,5.850,149.334
C03224=1164.129,-87.990,-42.682,179.021,5.851,149.334
C03225=1164.123,-87.740,-42.692,179.023,5.850,149.333
C03226=1164.117,-87.490,-42.702,179.025,5.851,149.332
C03227=1164.112,-87.241,-42.711,179.028,5.852,149.332
C03228=1164.107,-86.991,-42.722,179.030,5.851,149.331
C03229=1164.101,-86.741,-42.732,179.032,5.852,149.331
C03230=1164.096,-86.491,-42.741,179.034,5.852,149.330
C03231=1164.091,-86.242,-42.751,179.036,5.852,149.330
C03232=1164.085,-85.992,-42.762,179.038,5.853,149.329
C03233=1164.081,-85.742,-42.772,179.040,5.853,149.328
C03234=1164.075,-85.492,-42.781,179.043,5.854,149.328
C03235=1164.070,-85.243,-42.791,179.045,5.854,149.327
C03236=1164.064,-84.993,-42.801,179.047,5.854,149.327
C03237=1164.060,-84.743,-42.811,179.049,5.854,149.326
C03238=1164.054,-84.494,-42.822,179.052,5.855,149.326
C03239=1164.048,-84.243,-42.831,179.053,5.855,149.325
C03240=1164.043,-83.994,-42.841,179.056,5.855,149.324
C03241=1164.038,-83.744,-42.851,179.058,5.856,149.324
C03242=1164.033,-83.494,-42.862,179.060,5.856,149.323
C03243=1164.027,-83.245,-42.872,179.062,5.857,149.323
C03244=1164.022,-82.996,-42.881,179.065,5.857,149.322
C03245=1164.017,-82.745,-42.891,179.067,5.857,149.321
C03246=1164.011,-82.495,-42.901,179.069,5.857,149.321
C03247=1164.006,-82.246,-42.912,179.072,5.858,149.320
C03248=1164.001,-81.996,-42.922,179.073,5.858,149.320
C03249=1163.996,-81.746,-42.932,179.076,5.859,149.319
C03250=1163.990,-81.497,-42.942,179.078,5.859,149.319
C03251=1163.985,-81.247,-42.952,179.080,5.859,149.318
C03252=1163.980,-80.997,-42.962,179.082,5.860,149.317
C03253=1163.975,-80.748,-42.972,179.085,5.860,149.317
C03254=1163.969,-80.498,-42.983,179.086,5.860,149.316
C03255=1163.964,-80.247,-42.993,179.089,5.860,149.316
C03256=1163.958,-79.998,-43.003,179.091,5.861,149.315
C03257=1163.953,-79.748,-43.012,179.093,5.861,149.315
C03258=1163.948,-79.498,-43.023,179.096,5.862,149.314
C03259=1163.943,-79.249,-43.033,179.098,5.862,149.313
C03260=1163.937,-78.999,-43.043,179.100,5.862,149.313
C03261=1163.932,-78.749,-43.054,179.102,5.863,149.312
C03262=1163.927,-78.499,-43.064,179.105,5.863,149.311
C03263=1163.922,-78.250,-43.074,179.106,5.863,149.311
C03264=1163.917,-78.000,-43.084,179.109,5.864,149.310
C03265=1163.911,-77.750,-43.094,179.111,5.864,149.310
C03266=1163.906,-77.501,-43.105,179.113,5.864,149.309
C03267=1163.901,-77.251,-43.115,179.115,5.865,149.309
C03268=1163.895,-77.001,-43.125,179.118,5.865,149.308
C03269=1163.889,-76.751,-43.136,179.120,5.866,149.307
C03270=1163.884,-76.480,-43.147,179.122,5.865,149.307
C03271=1163.878,-76.209,-43.158,179.125,5.866,149.306
C03272=1163.873,-75.938,-43.169,179.127,5.867,149.306
C03273=1163.867,-75.667,-43.181,179.130,5.867,149.305
C03274=1163.861,-75.417,-43.191,179.132,5.868,149.304
C03275=1163.856,-75.167,-43.202,179.134,5.867,149.304
C03276=1163.851,-74.918,-43.211,179.136,5.868,149.303
C03277=1163.846,-74.668,-43.222,179.139,5.869,149.303
C03278=1163.841,-74.418,-43.232,179.141,5.869,149.302
C03279=1163.835,-74.169,-43.242,179.143,5.869,149.301
C03280=1163.830,-73.918,-43.253,179.146,5.870,149.301
C03281=1163.825,-73.669,-43.263,179.147,5.870,149.300
C03282=1163.819,-73.419,-43.273,179.150,5.870,149.300
C03283=1163.814,-73.170,-43.285,179.152,5.871,149.299
C03284=1163.809,-72.920,-43.295,179.155,5.871,149.298
C03285=1163.804,-72.670,-43.305,179.156,5.871,149.298
C03286=1163.798,-72.420,-43.316,179.159,5.872,149.297
C03287=1163.793,-72.171,-43.326,179.161,5.872,149.297
C03288=1163.788,-71.921,-43.336,179.163,5.872,149.296
C03289=1163.782,-71.671,-43.347,179.165,5.873,149.296
C03290=1163.777,-71.421,-43.358,179.168,5.873,149.295
C03291=1163.772,-71.172,-43.368,179.170,5.873,149.294
C03292=1163.766,-70.922,-43.378,179.172,5.874,149.294
C03293=1163.761,-70.672,-43.389,179.175,5.874,149.293
C03294=1163.756,-70.422,-43.399,179.177,5.875,149.293
C03295=1163.751,-70.173,-43.410,179.179,5.875,149.292
C03296=1163.745,-69.923,-43.421,179.181,5.876,149.291
C03297=1163.740,-69.673,-43.431,179.184,5.876,149.291
C03298=1163.735,-69.424,-43.441,179.185,5.876,149.290
C03299=1163.730,-69.174,-43.453,179.188,5.876,149.290
C03300=1163.724,-68.924,-43.463,179.190,5.877,149.289
C03301=1163.719,-68.674,-43.473,179.193,5.878,149.288
C03302=1163.714,-68.425,-43.484,179.194,5.878,149.288
C03303=1163.708,-68.176,-43.495,179.197,5.878,149.287
C03304=1163.703,-67.925,-43.505,179.199,5.879,149.287
C03305=1163.698,-67.676,-43.515,179.202,5.879,149.286
C03306=1163.693,-67.426,-43.526,179.203,5.879,149.286
C03307=1163.688,-67.177,-43.537,179.206,5.880,149.285
C03308=1163.683,-66.926,-43.547,179.208,5.880,149.284
C03309=1163.677,-66.677,-43.558,179.210,5.880,149.284
C03310=1163.672,-66.427,-43.569,179.213,5.881,149.283
C03311=1163.666,-66.177,-43.580,179.215,5.881,149.282
C03312=1163.661,-65.927,-43.590,179.217,5.882,149.282
C03313=1163.656,-65.678,-43.601,179.220,5.881,149.281
C03314=1163.651,-65.428,-43.612,179.222,5.882,149.281
C03315=1163.645,-65.178,-43.622,179.224,5.883,149.280
C03316=1163.640,-64.929,-43.633,179.227,5.883,149.280
C03317=1163.635,-64.679,-43.644,179.229,5.883,149.279
C03318=1163.630,-64.430,-43.655,179.231,5.884,149.278
C03319=1163.624,-64.180,-43.665,179.234,5.884,149.278
C03320=1163.619,-63.930,-43.676,179.236,5.885,149.277
C03321=1163.614,-63.680,-43.688,179.238,5.885,149.277
C03322=1163.608,-63.430,-43.698,179.240,5.885,149.276
C03323=1163.604,-63.181,-43.709,179.243,5.886,149.275
C03324=1163.598,-62.931,-43.719,179.245,5.887,149.275
C03325=1163.593,-62.681,-43.730,179.247,5.886,149.274
C03326=1163.588,-62.432,-43.741,179.249,5.887,149.274
C03327=1163.582,-62.182,-43.752,179.252,5.887,149.273
C03328=1163.577,-61.933,-43.763,179.254,5.888,149.272
C03329=1163.572,-61.682,-43.773,179.256,5.888,149.272
C03330=1163.567,-61.433,-43.785,179.258,5.889,149.271
C03331=1163.562,-61.183,-43.795,179.261,5.889,149.271
C03332=1163.556,-60.933,-43.807,179.263,5.890,149.270
C03333=1163.551,-60.684,-43.817,179.265,5.889,149.269
C03334=1163.546,-60.434,-43.828,179.267,5.890,149.269
C03335=1163.540,-60.185,-43.838,179.270,5.891,149.268
C03336=1163.536,-59.935,-43.850,179.272,5.891,149.268
C03337=1163.530,-59.684,-43.861,179.274,5.891,149.267
C03338=1163.525,-59.435,-43.872,179.276,5.892,149.267
C03339=1163.520,-59.185,-43.882,179.279,5.892,149.266
C03340=1163.515,-58.936,-43.894,179.281,5.893,149.265
C03341=1163.509,-58.686,-43.904,179.284,5.893,149.265
C03342=1163.504,-58.436,-43.916,179.286,5.893,149.264
C03343=1163.499,-58.187,-43.927,179.288,5.894,149.264
C03344=1163.494,-57.937,-43.937,179.290,5.895,149.263
C03345=1163.489,-57.687,-43.949,179.293,5.895,149.262
C03346=1163.482,-57.437,-43.959,179.295,5.895,149.262
C03347=1163.478,-57.188,-43.971,179.297,5.895,149.261
C03348=1163.473,-56.938,-43.982,179.300,5.896,149.261
C03349=1163.467,-56.689,-43.992,179.302,5.897,149.260
C03350=1163.462,-56.439,-44.004,179.304,5.897,149.259
C03351=1163.456,-56.189,-44.014,179.306,5.897,149.259
C03352=1163.452,-55.940,-44.026,179.309,5.898,149.258
C03353=1163.446,-55.690,-44.037,179.311,5.898,149.258
C03354=1163.441,-55.440,-44.048,179.313,5.899,149.257
C03355=1163.436,-55.190,-44.059,179.316,5.899,149.256
C03356=1163.431,-54.940,-44.071,179.318,5.899,149.256
C03357=1163.425,-54.691,-44.081,179.320,5.900,149.255
C03358=1163.420,-54.441,-44.092,179.323,5.901,149.255
C03359=1163.415,-54.191,-44.104,179.325,5.901,149.254
C03360=1163.409,-53.942,-44.114,179.327,5.901,149.253
C03361=1163.405,-53.692,-44.126,179.330,5.901,149.253
C03362=1163.399,-53.442,-44.138,179.332,5.902,149.252
C03363=1163.394,-53.192,-44.148,179.334,5.903,149.252
C03364=1163.389,-52.943,-44.159,179.337,5.903,149.251
C03365=1163.383,-52.693,-44.171,179.339,5.903,149.251
C03366=1163.379,-52.444,-44.182,179.341,5.903,149.250
C03367=1163.373,-52.194,-44.193,179.343,5.904,149.249
C03368=1163.368,-51.944,-44.204,179.346,5.905,149.249
C03369=1163.363,-51.694,-44.216,179.348,5.905,149.248
C03370=1163.357,-51.445,-44.227,179.350,5.905,149.247
C03371=1163.352,-51.195,-44.238,179.353,5.906,149.247
C03372=1163.347,-50.945,-44.249,179.355,5.906,149.246
C03373=1163.342,-50.695,-44.261,179.357,5.907,149.246
C03374=1163.336,-50.425,-44.273,179.360,5.907,149.245
C03375=1163.331,-50.155,-44.285,179.363,5.908,149.244
C03376=1163.325,-49.885,-44.297,179.365,5.908,149.244
C03377=1163.319,-49.614,-44.309,179.368,5.909,149.243
C03378=1163.314,-49.364,-44.321,179.370,5.909,149.242
C03379=1163.309,-49.114,-44.333,179.372,5.910,149.242
C03380=1163.303,-48.865,-44.344,179.375,5.910,149.241
C03381=1163.298,-48.615,-44.355,179.377,5.911,149.241
C03382=1163.293,-48.365,-44.367,179.379,5.911,149.240
C03383=1163.288,-48.115,-44.378,179.382,5.912,149.240
C03384=1163.282,-47.866,-44.389,179.384,5.912,149.239
C03385=1163.277,-47.616,-44.401,179.386,5.912,149.238
C03386=1163.273,-47.367,-44.412,179.389,5.913,149.238
C03387=1163.267,-47.117,-44.424,179.391,5.913,149.237
C03388=1163.262,-46.868,-44.435,179.393,5.914,149.237
C03389=1163.256,-46.618,-44.447,179.396,5.914,149.236
C03390=1163.251,-46.368,-44.457,179.398,5.914,149.235
C03391=1163.246,-46.118,-44.469,179.400,5.915,149.235
C03392=1163.241,-45.868,-44.481,179.402,5.916,149.234
C03393=1163.235,-45.619,-44.492,179.405,5.916,149.234
C03394=1163.230,-45.369,-44.504,179.407,5.917,149.233
C03395=1163.225,-45.119,-44.515,179.410,5.917,149.232
C03396=1163.220,-44.869,-44.527,179.412,5.917,149.232
C03397=1163.215,-44.620,-44.538,179.414,5.918,149.231
C03398=1163.209,-44.371,-44.550,179.416,5.918,149.231
C03399=1163.204,-44.121,-44.561,179.419,5.919,149.230
C03400=1163.199,-43.871,-44.573,179.422,5.919,149.229
C03401=1163.194,-43.621,-44.584,179.424,5.920,149.229
C03402=1163.189,-43.371,-44.596,179.426,5.920,149.228
C03403=1163.183,-43.122,-44.608,179.428,5.921,149.228
C03404=1163.178,-42.873,-44.619,179.431,5.921,149.227
C03405=1163.173,-42.623,-44.631,179.433,5.922,149.226
C03406=1163.168,-42.373,-44.642,179.436,5.922,149.226
C03407=1163.163,-42.123,-44.654,179.438,5.923,149.225
C03408=1163.158,-41.873,-44.665,179.441,5.923,149.225
C03409=1163.152,-41.623,-44.677,179.442,5.923,149.224
C03410=1163.146,-41.374,-44.689,179.445,5.924,149.223
C03411=1163.142,-41.125,-44.700,179.447,5.925,149.223
C03412=1163.137,-40.875,-44.713,179.450,5.925,149.222
C03413=1163.131,-40.625,-44.724,179.452,5.925,149.222
C03414=1163.126,-40.376,-44.736,179.455,5.926,149.221
C03415=1163.121,-40.126,-44.748,179.457,5.927,149.220
C03416=1163.116,-39.876,-44.759,179.459,5.927,149.220
C03417=1163.111,-39.626,-44.771,179.461,5.927,149.219
C03418=1163.105,-39.377,-44.782,179.464,5.928,149.219
C03419=1163.099,-39.127,-44.794,179.466,5.928,149.218
C03420=1163.095,-38.878,-44.806,179.468,5.929,149.218
C03421=1163.090,-38.628,-44.818,179.471,5.930,149.217
C03422=1163.084,-38.378,-44.830,179.473,5.930,149.216
C03423=1163.079,-38.129,-44.841,179.475,5.930,149.216
C03424=1163.074,-37.879,-44.853,179.478,5.930,149.215
C03425=1163.069,-37.629,-44.865,179.480,5.931,149.215
C03426=1163.064,-37.380,-44.877,179.483,5.932,149.214
C03427=1163.058,-37.130,-44.889,179.485,5.932,149.213
C03428=1163.053,-36.881,-44.900,179.488,5.933,149.213
C03429=1163.047,-36.631,-44.912,179.490,5.934,149.212
C03430=1163.043,-36.381,-44.924,179.493,5.934,149.211
C03431=1163.038,-36.132,-44.936,179.494,5.934,149.211
C03432=1163.032,-35.882,-44.948,179.497,5.934,149.210
C03433=1163.027,-35.632,-44.959,179.499,5.935,149.210
C03434=1163.022,-35.382,-44.971,179.502,5.936,149.209
C03435=1163.017,-35.133,-44.984,179.504,5.936,149.208
C03436=1163.011,-34.883,-44.996,179.507,5.937,149.208
C03437=1163.007,-34.633,-45.007,179.509,5.937,149.207
C03438=1163.001,-34.383,-45.019,179.511,5.938,149.207
C03439=1162.996,-34.134,-45.032,179.514,5.939,149.206
C03440=1162.991,-33.884,-45.043,179.516,5.939,149.206
C03441=1162.985,-33.634,-45.055,179.518,5.939,149.205
C03442=1162.981,-33.385,-45.067,179.520,5.940,149.204
C03443=1162.975,-33.135,-45.079,179.523,5.940,149.204
C03444=1162.970,-32.885,-45.091,179.526,5.941,149.203
C03445=1162.965,-32.636,-45.104,179.528,5.941,149.203
C03446=1162.960,-32.386,-45.116,179.531,5.942,149.202
C03447=1162.955,-32.136,-45.127,179.533,5.943,149.201
C03448=1162.950,-31.887,-45.139,179.535,5.943,149.201
C03449=1162.944,-31.637,-45.151,179.538,5.944,149.200
C03450=1162.939,-31.387,-45.163,179.540,5.944,149.200
C03451=1162.934,-31.138,-45.176,179.542,5.944,149.199
C03452=1162.928,-30.888,-45.188,179.545,5.945,149.198
C03453=1162.924,-30.639,-45.200,179.547,5.946,149.198
C03454=1162.918,-30.389,-45.212,179.549,5.946,149.197
C03455=1162.913,-30.139,-45.223,179.552,5.946,149.196
C03456=1162.908,-29.890,-45.236,179.554,5.947,149.196
C03457=1162.902,-29.640,-45.248,179.557,5.948,149.195
C03458=1162.897,-29.390,-45.261,179.559,5.948,149.195
C03459=1162.892,-29.141,-45.272,179.562,5.949,149.194
C03460=1162.887,-28.891,-45.285,179.564,5.950,149.194
C03461=1162.882,-28.642,-45.296,179.567,5.950,149.193
C03462=1162.877,-28.392,-45.309,179.568,5.950,149.193
C03463=1162.872,-28.142,-45.321,179.571,5.951,149.192
C03464=1162.866,-27.893,-45.333,179.574,5.951,149.191
C03465=1162.861,-27.643,-45.345,179.576,5.952,149.191
C03466=1162.856,-27.394,-45.358,179.578,5.952,149.190
C03467=1162.850,-27.144,-45.370,179.581,5.953,149.189
C03468=1162.845,-26.895,-45.382,179.583,5.954,149.189
C03469=1162.840,-26.645,-45.394,179.585,5.954,149.188
C03470=1162.835,-26.395,-45.407,179.588,5.955,149.188
C03471=1162.830,-26.145,-45.419,179.590,5.956,149.187
C03472=1162.825,-25.895,-45.432,179.593,5.956,149.186
C03473=1162.819,-25.645,-45.444,179.596,5.956,149.186
C03474=1162.815,-25.396,-45.456,179.598,5.957,149.185
C03475=1162.810,-25.146,-45.468,179.600,5.958,149.185
C03476=1162.804,-24.897,-45.480,179.603,5.958,149.184
C03477=1162.799,-24.648,-45.493,179.605,5.958,149.183
C03478=1162.793,-24.377,-45.506,179.608,5.959,149.183
C03479=1162.788,-24.107,-45.520,179.610,5.960,149.182
C03480=1162.782,-23.838,-45.533,179.613,5.961,149.182
C03481=1162.777,-23.568,-45.547,179.615,5.961,149.181
C03482=1162.771,-23.318,-45.559,179.618,5.962,149.180
C03483=1162.766,-23.068,-45.571,179.620,5.962,149.180
C03484=1162.761,-22.819,-45.584,179.623,5.963,149.179
C03485=1162.756,-22.569,-45.596,179.625,5.963,149.179
C03486=1162.751,-22.319,-45.609,179.628,5.964,149.178
C03487=1162.746,-22.070,-45.621,179.630,5.965,149.177
C03488=1162.740,-21.820,-45.633,179.633,5.965,149.177
C03489=1162.735,-21.571,-45.646,179.635,5.966,149.176
C03490=1162.730,-21.321,-45.658,179.637,5.966,149.175
C03491=1162.725,-21.071,-45.670,179.639,5.966,149.175
C03492=1162.720,-20.822,-45.683,179.642,5.967,149.174
C03493=1162.715,-20.572,-45.696,179.644,5.967,149.174
C03494=1162.710,-20.322,-45.708,179.647,5.968,149.173
C03495=1162.705,-20.073,-45.720,179.649,5.969,149.172
C03496=1162.699,-19.823,-45.734,179.651,5.969,149.172
C03497=1162.694,-19.574,-45.746,179.654,5.970,149.171
C03498=1162.688,-19.324,-45.758,179.656,5.971,149.171
C03499=1162.684,-19.074,-45.771,179.659,5.971,149.170
C03500=1162.679,-18.825,-45.784,179.662,5.971,149.169
C03501=1162.673,-18.575,-45.796,179.664,5.972,149.169
C03502=1162.668,-18.326,-45.809,179.666,5.973,149.168
C03503=1162.663,-18.076,-45.821,179.669,5.974,149.168
C03504=1162.658,-17.826,-45.834,179.671,5.974,149.167
C03505=1162.652,-17.576,-45.847,179.673,5.975,149.167
C03506=1162.647,-17.327,-45.859,179.676,5.975,149.166
C03507=1162.642,-17.078,-45.872,179.678,5.976,149.165
C03508=1162.638,-16.828,-45.885,179.681,5.976,149.165
C03509=1162.632,-16.578,-45.897,179.684,5.977,149.164
C03510=1162.626,-16.328,-45.910,179.686,5.978,149.164
C03511=1162.621,-16.079,-45.923,179.688,5.978,149.163
C03512=1162.616,-15.829,-45.935,179.691,5.979,149.162
C03513=1162.612,-15.579,-45.948,179.693,5.979,149.162
C03514=1162.607,-15.330,-45.961,179.695,5.980,149.161
C03515=1162.601,-15.081,-45.974,179.698,5.981,149.161
C03516=1162.596,-14.831,-45.987,179.700,5.981,149.160
C03517=1162.591,-14.581,-45.999,179.703,5.982,149.159
C03518=1162.586,-14.331,-46.012,179.706,5.982,149.159
C03519=1162.580,-14.082,-46.024,179.708,5.983,149.158
C03520=1162.575,-13.832,-46.038,179.710,5.984,149.158
C03521=1162.570,-13.582,-46.050,179.713,5.984,149.157
C03522=1162.565,-13.333,-46.063,179.715,5.985,149.156
C03523=1162.560,-13.084,-46.076,179.717,5.986,149.156
C03524=1162.555,-12.833,-46.089,179.720,5.986,149.155
C03525=1162.549,-12.584,-46.102,179.723,5.987,149.155
C03526=1162.544,-12.335,-46.114,179.725,5.987,149.154
C03527=1162.540,-12.085,-46.127,179.728,5.988,149.153
C03528=1162.534,-11.835,-46.140,179.730,5.989,149.153
C03529=1162.529,-11.586,-46.153,179.732,5.989,149.152
C03530=1162.524,-11.336,-46.166,179.735,5.990,149.152
C03531=1162.519,-11.086,-46.179,179.737,5.990,149.151
C03532=1162.513,-10.837,-46.192,179.739,5.991,149.151
C03533=1162.508,-10.587,-46.204,179.742,5.992,149.150
C03534=1162.504,-10.337,-46.217,179.745,5.992,149.149
C03535=1162.498,-10.088,-46.231,179.747,5.993,149.149
C03536=1162.493,-9.838,-46.243,179.750,5.993,149.148
C03537=1162.488,-9.588,-46.256,179.752,5.994,149.148
C03538=1162.483,-9.339,-46.270,179.754,5.995,149.147
C03539=1162.478,-9.089,-46.283,179.757,5.995,149.146
C03540=1162.473,-8.840,-46.296,179.759,5.996,149.146
C03541=1162.467,-8.590,-46.309,179.762,5.996,149.145
C03542=1162.463,-8.340,-46.322,179.764,5.997,149.145
C03543=1162.457,-8.091,-46.334,179.767,5.998,149.144
C03544=1162.452,-7.841,-46.348,179.769,5.998,149.143
C03545=1162.447,-7.591,-46.361,179.772,6.000,149.143
C03546=1162.441,-7.342,-46.374,179.774,6.000,149.142
C03547=1162.436,-7.093,-46.387,179.777,6.001,149.142
C03548=1162.432,-6.843,-46.400,179.779,6.002,149.141
C03549=1162.426,-6.594,-46.413,179.782,6.002,149.140
C03550=1162.421,-6.343,-46.426,179.784,6.003,149.140
C03551=1162.416,-6.094,-46.439,179.787,6.003,149.139
C03552=1162.411,-5.845,-46.453,179.789,6.004,149.139
C03553=1162.406,-5.595,-46.466,179.791,6.005,149.138
C03554=1162.400,-5.346,-46.479,179.794,6.005,149.137
C03555=1162.396,-5.095,-46.492,179.796,6.006,149.137
C03556=1162.390,-4.846,-46.506,179.799,6.006,149.136
C03557=1162.385,-4.597,-46.518,179.802,6.007,149.136
C03558=1162.380,-4.347,-46.532,179.804,6.008,149.135
C03559=1162.375,-4.098,-46.545,179.806,6.008,149.134
C03560=1162.370,-3.848,-46.559,179.809,6.009,149.134
C03561=1162.365,-3.598,-46.571,179.811,6.009,149.133
C03562=1162.360,-3.348,-46.584,179.813,6.010,149.133
C03563=1162.354,-3.099,-46.598,179.816,6.011,149.132
C03564=1162.350,-2.850,-46.611,179.818,6.011,149.132
C03565=1162.344,-2.600,-46.624,179.821,6.013,149.131
C03566=1162.339,-2.351,-46.637,179.824,6.013,149.130
C03567=1162.334,-2.101,-46.651,179.826,6.014,149.130
C03568=1162.329,-1.851,-46.664,179.829,6.014,149.129
C03569=1162.324,-1.601,-46.677,179.831,6.015,149.129
C03570=1162.318,-1.352,-46.691,179.834,6.016,149.128
C03571=1162.314,-1.102,-46.704,179.836,6.017,149.128
C03572=1162.308,-0.852,-46.718,179.839,6.017,149.127
C03573=1162.304,-0.603,-46.731,179.841,6.018,149.126
C03574=1162.298,-0.353,-46.744,179.843,6.018,149.126
C03575=1162.294,-0.104,-46.758,179.846,6.019,149.125
C03576=1162.288,0.146,-46.771,179.848,6.020,149.125
C03577=1162.283,0.396,-46.784,179.851,6.020,149.124
C03578=1162.278,0.645,-46.798,179.854,6.022,149.123
C03579=1162.272,0.895,-46.812,179.856,6.022,149.123
C03580=1162.268,1.144,-46.825,179.859,6.023,149.122
C03581=1162.262,1.394,-46.839,179.861,6.023,149.122
C03582=1162.257,1.662,-46.853,179.864,6.024,149.121
C03583=1162.252,1.932,-46.868,179.866,6.025,149.120
C03584=1162.246,2.202,-46.882,179.869,6.026,149.120
C03585=1162.240,2.471,-46.897,179.872,6.026,149.119
C03586=1162.235,2.721,-46.909,179.875,6.027,149.118
C03587=1162.230,2.970,-46.924,179.877,6.028,149.118
C03588=1162.224,3.220,-46.937,179.879,6.028,149.117
C03589=1162.220,3.469,-46.951,179.882,6.029,149.117
C03590=1162.214,3.719,-46.964,179.884,6.029,149.116
C03591=1162.209,3.969,-46.978,179.886,6.030,149.116
C03592=1162.205,4.217,-46.991,179.890,6.031,149.115
C03593=1162.199,4.468,-47.005,179.892,6.032,149.114
C03594=1162.194,4.717,-47.019,179.894,6.033,149.114
C03595=1162.189,4.967,-47.032,179.897,6.033,149.113
C03596=1162.184,5.216,-47.046,179.899,6.034,149.113
C03597=1162.178,5.466,-47.059,179.902,6.034,149.112
C03598=1162.174,5.715,-47.073,179.904,6.035,149.111
C03599=1162.169,5.964,-47.087,179.907,6.036,149.111
C03600=1162.163,6.215,-47.101,179.909,6.037,149.110
C03601=1162.159,6.464,-47.114,179.912,6.038,149.110
C03602=1162.153,6.714,-47.127,179.914,6.039,149.109
C03603=1162.148,6.964,-47.142,179.917,6.039,149.108
C03604=1162.143,7.213,-47.156,179.920,6.040,149.108
C03605=1162.138,7.463,-47.169,179.922,6.040,149.107
C03606=1162.133,7.712,-47.183,179.924,6.041,149.107
C03607=1162.128,7.961,-47.197,179.927,6.042,149.106
C03608=1162.123,8.212,-47.210,179.929,6.042,149.105
C03609=1162.118,8.460,-47.224,179.932,6.044,149.105
C03610=1162.113,8.710,-47.238,179.935,6.044,149.104
C03611=1162.107,8.960,-47.251,179.937,6.045,149.104
C03612=1162.102,9.209,-47.265,179.940,6.046,149.103
C03613=1162.098,9.459,-47.279,179.942,6.046,149.103
C03614=1162.093,9.708,-47.293,179.944,6.047,149.102
C03615=1162.087,9.958,-47.307,179.947,6.047,149.101
C03616=1162.082,10.208,-47.321,179.950,6.049,149.101
C03617=1162.077,10.457,-47.335,179.952,6.049,149.100
C03618=1162.071,10.706,-47.349,179.955,6.050,149.100
C03619=1162.067,10.957,-47.362,179.957,6.051,149.099
C03620=1162.062,11.206,-47.376,179.959,6.051,149.099
C03621=1162.056,11.455,-47.390,179.962,6.052,149.098
C03622=1162.051,11.705,-47.404,179.964,6.053,149.097
C03623=1162.046,11.955,-47.419,179.967,6.054,149.097
C03624=1162.041,12.204,-47.432,179.970,6.054,149.096
C03625=1162.036,12.454,-47.446,179.972,6.055,149.096
C03626=1162.031,12.703,-47.460,179.975,6.056,149.095
C03627=1162.026,12.952,-47.474,179.977,6.057,149.095
C03628=1162.021,13.202,-47.488,179.980,6.057,149.094
C03629=1162.016,13.452,-47.502,179.983,6.059,149.093
C03630=1162.011,13.702,-47.516,179.985,6.059,149.093
C03631=1162.005,13.951,-47.530,179.987,6.060,149.092
C03632=1162.000,14.201,-47.544,179.990,6.060,149.092
C03633=1161.996,14.450,-47.558,179.992,6.061,149.091
C03634=1161.990,14.699,-47.572,179.995,6.062,149.090
C03635=1161.985,14.949,-47.586,179.997,6.062,149.090
C03636=1161.981,15.199,-47.600,-180.000,6.064,149.089
C03637=1161.976,15.448,-47.614,-179.997,6.064,149.089
C03638=1161.970,15.697,-47.628,-179.995,6.065,149.088
C03639=1161.965,15.947,-47.643,-179.992,6.066,149.087
C03640=1161.960,16.197,-47.657,-179.990,6.066,149.087
C03641=1161.955,16.447,-47.671,-179.987,6.068,149.086
C03642=1161.949,16.696,-47.684,-179.985,6.069,149.086
C03643=1161.944,16.946,-47.699,-179.982,6.069,149.085
C03644=1161.939,17.196,-47.713,-179.980,6.070,149.085
C03645=1161.934,17.445,-47.727,-179.977,6.070,149.084
C03646=1161.929,17.694,-47.741,-179.975,6.071,149.083
C03647=1161.924,17.944,-47.755,-179.972,6.072,149.083
C03648=1161.919,18.194,-47.770,-179.969,6.073,149.082
C03649=1161.914,18.443,-47.785,-179.967,6.074,149.082
C03650=1161.909,18.693,-47.799,-179.964,6.074,149.081
C03651=1161.904,18.942,-47.813,-179.962,6.075,149.081
C03652=1161.899,19.191,-47.827,-179.959,6.076,149.080
C03653=1161.894,19.441,-47.841,-179.957,6.077,149.079
C03654=1161.889,19.691,-47.856,-179.954,6.078,149.079
C03655=1161.884,19.940,-47.870,-179.952,6.078,149.078
